LIN {X 0,Y 573.33,Z 232.072,A -85,B 0,C 180,E1 -2340.702,E2 -2340.702} C_VEL
LIN {X 0,Y 573.232,Z 232.084,A -85,B 0,C 180,E1 -2343.514,E2 -2343.514} C_VEL
LIN {X 0,Y 573.285,Z 232.078,A -85,B 0,C 180,E1 -2345.627,E2 -2345.627} C_VEL
LIN {X 0,Y 573.302,Z 232.075,A -85,B 0,C 180,E1 -2348.458,E2 -2348.458} C_VEL
LIN {X 0,Y 573.232,Z 232.085,A -85,B 0,C 180,E1 -2350.596,E2 -2350.596} C_VEL
LIN {X 0,Y 573.186,Z 234.19,A -85,B 0,C 180,E1 -2352.03,E2 -2352.03} C_VEL
LIN {X 0,Y 573.193,Z 239.014,A -85,B 0,C 180,E1 -2354.92,E2 -2354.92} C_VEL
LIN {X 0,Y 573.132,Z 244.034,A -85,B 0,C 180,E1 -2357.851,E2 -2357.851} C_VEL
LIN {X 0,Y 573.107,Z 249.239,A -85,B 0,C 180,E1 -2360.831,E2 -2360.831} C_VEL
LIN {X 0,Y 573.09,Z 253.122,A -85,B 0,C 180,E1 -2363.113,E2 -2363.113} C_VEL
LIN {X 0,Y 573.02,Z 254.947,A -85,B 0,C 180,E1 -2364.165,E2 -2364.165} C_VEL
LIN {X 0,Y 572.332,Z 256.016,A -85,B 0,C 180,E1 -2364.741,E2 -2364.741} C_VEL
LIN {X 0,Y 569.439,Z 257.913,A -85,B 0,C 180,E1 -2365.674,E2 -2365.674} C_VEL
LIN {X 0,Y 567.014,Z 259.45,A -85,B 0,C 180,E1 -2366.423,E2 -2366.423} C_VEL
LIN {X 0,Y 565.992,Z 260.576,A -85,B 0,C 180,E1 -2367.003,E2 -2367.003} C_VEL
LIN {X 0,Y 565.919,Z 260.939,A -85,B 0,C 180,E1 -2367.2,E2 -2367.2} C_VEL
LIN {X 0,Y 565.873,Z 265.731,A -85,B 0,C 180,E1 -2369.787,E2 -2369.787} C_VEL
LIN {X 0,Y 565.858,Z 270.593,A -85,B 0,C 180,E1 -2372.377,E2 -2372.377} C_VEL
LIN {X 0,Y 565.894,Z 272.598,A -85,B 0,C 180,E1 -2373.417,E2 -2373.417} C_VEL
LIN {X 0,Y 566.93,Z 280.016,A -85,B 0,C 180,E1 -2373.598,E2 -2373.598} C_VEL
LIN {X 0,Y 566.775,Z 292.555,A -85,B 0,C 180,E1 -2373.97,E2 -2373.97} C_VEL
LIN {X 0,Y 566.643,Z 304.455,A -85,B 0,C 180,E1 -2374.462,E2 -2374.462} C_VEL
LIN {X 0,Y 566.533,Z 315.205,A -85,B 0,C 180,E1 -2375.042,E2 -2375.042} C_VEL
LIN {X 0,Y 566.409,Z 325.926,A -85,B 0,C 180,E1 -2375.771,E2 -2375.771} C_VEL
LIN {X 0,Y 566.276,Z 336.609,A -85,B 0,C 180,E1 -2376.674,E2 -2376.674} C_VEL
LIN {X 0,Y 566.178,Z 344.253,A -85,B 0,C 180,E1 -2377.461,E2 -2377.461} C_VEL
LIN {X 0,Y 566.028,Z 352.881,A -85,B 0,C 180,E1 -2378.536,E2 -2378.536} C_VEL
LIN {X 0,Y 565.982,Z 360.04,A -85,B 0,C 180,E1 -2379.659,E2 -2379.659} C_VEL
LIN {X 0,Y 565.939,Z 365.613,A -85,B 0,C 180,E1 -2380.756,E2 -2380.756} C_VEL
LIN {X 0,Y 565.92,Z 369.886,A -85,B 0,C 180,E1 -2381.832,E2 -2381.832} C_VEL
LIN {X 0,Y 565.849,Z 373.537,A -85,B 0,C 180,E1 -2383.086,E2 -2383.086} C_VEL
LIN {X 0,Y 565.854,Z 375.448,A -85,B 0,C 180,E1 -2384.068,E2 -2384.068} C_VEL
LIN {X 0,Y 565.874,Z 376.606,A -85,B 0,C 180,E1 -2385.065,E2 -2385.065} C_VEL
LIN {X 0,Y 565.845,Z 376.997,A -85,B 0,C 180,E1 -2386.084,E2 -2386.084} C_VEL
LIN {X 0,Y 565.846,Z 376.542,A -85,B 0,C 180,E1 -2387.12,E2 -2387.12} C_VEL
LIN {X 0,Y 565.851,Z 375.204,A -85,B 0,C 180,E1 -2388.176,E2 -2388.176} C_VEL
LIN {X 0,Y 565.869,Z 372.917,A -85,B 0,C 180,E1 -2389.252,E2 -2389.252} C_VEL
LIN {X 0,Y 565.945,Z 369.582,A -85,B 0,C 180,E1 -2390.345,E2 -2390.345} C_VEL
LIN {X 0,Y 565.942,Z 364.323,A -85,B 0,C 180,E1 -2391.618,E2 -2391.618} C_VEL
LIN {X 0,Y 566.024,Z 357.686,A -85,B 0,C 180,E1 -2392.828,E2 -2392.828} C_VEL
LIN {X 0,Y 566.066,Z 351.029,A -85,B 0,C 180,E1 -2393.802,E2 -2393.802} C_VEL
LIN {X 0,Y 566.178,Z 342.022,A -85,B 0,C 180,E1 -2394.876,E2 -2394.876} C_VEL
LIN {X 0,Y 566.32,Z 331.919,A -85,B 0,C 180,E1 -2395.838,E2 -2395.838} C_VEL
LIN {X 0,Y 566.432,Z 320.626,A -85,B 0,C 180,E1 -2396.7,E2 -2396.7} C_VEL
LIN {X 0,Y 566.531,Z 308.684,A -85,B 0,C 180,E1 -2397.416,E2 -2397.416} C_VEL
LIN {X 0,Y 566.702,Z 296.228,A -85,B 0,C 180,E1 -2397.984,E2 -2397.984} C_VEL
LIN {X 0,Y 566.865,Z 283.269,A -85,B 0,C 180,E1 -2398.412,E2 -2398.412} C_VEL
LIN {X 0,Y 566.692,Z 277.469,A -85,B 0,C 180,E1 -2398.558,E2 -2398.558} C_VEL
LIN {X 0,Y 565.854,Z 272.554,A -85,B 0,C 180,E1 -2398.677,E2 -2398.677} C_VEL
LIN {X 0,Y 565.849,Z 268.118,A -85,B 0,C 180,E1 -2401.028,E2 -2401.028} C_VEL
LIN {X 0,Y 565.887,Z 263.61,A -85,B 0,C 180,E1 -2403.443,E2 -2403.443} C_VEL
LIN {X 0,Y 565.906,Z 259.28,A -85,B 0,C 180,E1 -2405.807,E2 -2405.807} C_VEL
LIN {X 0,Y 565.967,Z 254.293,A -85,B 0,C 180,E1 -2408.639,E2 -2408.639} C_VEL
LIN {X 0,Y 566.028,Z 249.915,A -85,B 0,C 180,E1 -2411.167,E2 -2411.167} C_VEL
LIN {X 0,Y 566.041,Z 244.734,A -85,B 0,C 180,E1 -2414.148,E2 -2414.148} C_VEL
LIN {X 0,Y 566.11,Z 239.77,A -85,B 0,C 180,E1 -2417.088,E2 -2417.088} C_VEL
LIN {X 0,Y 566.19,Z 236.152,A -85,B 0,C 180,E1 -2419.27,E2 -2419.27} C_VEL
LIN {X 0,Y 566.131,Z 233.791,A -85,B 0,C 180,E1 -2420.713,E2 -2420.713} C_VEL
LIN {X 0,Y 566.158,Z 232.962,A -85,B 0,C 180,E1 -2421.434,E2 -2421.434} C_VEL
LIN {X 0,Y 566.197,Z 232.961,A -85,B 0,C 180,E1 -2423.586,E2 -2423.586} C_VEL
LIN {X 0,Y 566.184,Z 232.96,A -85,B 0,C 180,E1 -2425.729,E2 -2425.729} C_VEL
LIN {X 0,Y 566.267,Z 232.949,A -85,B 0,C 180,E1 -2427.866,E2 -2427.866} C_VEL
LIN {X 0,Y 566.297,Z 232.948,A -85,B 0,C 180,E1 -2430.711,E2 -2430.711} C_VEL
LIN {X 0,Y 566.267,Z 232.95,A -85,B 0,C 180,E1 -2432.846,E2 -2432.846} C_VEL
LIN {X 0,Y 566.251,Z 232.954,A -85,B 0,C 180,E1 -2435.698,E2 -2435.698} C_VEL
LIN {X 0,Y 566.241,Z 232.953,A -85,B 0,C 180,E1 -2438.565,E2 -2438.565} C_VEL
LIN {X 0,Y 566.24,Z 232.954,A -85,B 0,C 180,E1 -2441.454,E2 -2441.454} C_VEL
LIN {X 0,Y 566.223,Z 232.955,A -85,B 0,C 180,E1 -2444.507,E2 -2444.507} C_VEL
LIN {X 0,Y 566.195,Z 232.959,A -85,B 0,C 180,E1 -2447.332,E2 -2447.332} C_VEL
LIN {X 0,Y 566.21,Z 232.957,A -85,B 0,C 180,E1 -2450.337,E2 -2450.337} C_VEL
LIN {X 0,Y 566.22,Z 232.956,A -85,B 0,C 180,E1 -2453.402,E2 -2453.402} C_VEL
LIN {X 0,Y 566.213,Z 232.957,A -85,B 0,C 180,E1 -2455.749,E2 -2455.749} C_VEL
LIN {X 0,Y 566.198,Z 232.96,A -85,B 0,C 180,E1 -2458.204,E2 -2458.204} C_VEL
LIN {X 0,Y 566.184,Z 232.961,A -85,B 0,C 180,E1 -2460.592,E2 -2460.592} C_VEL
LIN {X 0,Y 566.218,Z 232.957,A -85,B 0,C 180,E1 -2463.102,E2 -2463.102} C_VEL
LIN {X 0,Y 566.201,Z 232.96,A -85,B 0,C 180,E1 -2465.689,E2 -2465.689} C_VEL
LIN {X 0,Y 566.207,Z 232.956,A -85,B 0,C 180,E1 -2468.56,E2 -2468.56} C_VEL
LIN {X 0,Y 566.201,Z 232.958,A -85,B 0,C 180,E1 -2471.136,E2 -2471.136} C_VEL
LIN {X 0,Y 566.189,Z 232.962,A -85,B 0,C 180,E1 -2474.036,E2 -2474.036} C_VEL
LIN {X 0,Y 566.202,Z 232.957,A -85,B 0,C 180,E1 -2477.082,E2 -2477.082} C_VEL
LIN {X 0,Y 566.216,Z 232.957,A -85,B 0,C 180,E1 -2479.803,E2 -2479.803} C_VEL
LIN {X 0,Y 566.188,Z 232.961,A -85,B 0,C 180,E1 -2482.599,E2 -2482.599} C_VEL
LIN {X 0,Y 566.209,Z 232.957,A -85,B 0,C 180,E1 -2485.184,E2 -2485.184} C_VEL
LIN {X 0,Y 566.225,Z 232.954,A -85,B 0,C 180,E1 -2487.744,E2 -2487.744} C_VEL
LIN {X 0,Y 566.217,Z 232.955,A -85,B 0,C 180,E1 -2490.324,E2 -2490.324} C_VEL
LIN {X 0,Y 566.225,Z 232.956,A -85,B 0,C 180,E1 -2493.336,E2 -2493.336} C_VEL
LIN {X 0,Y 566.19,Z 232.96,A -85,B 0,C 180,E1 -2495.82,E2 -2495.82} C_VEL
LIN {X 0,Y 566.208,Z 232.958,A -85,B 0,C 180,E1 -2498.903,E2 -2498.903} C_VEL
LIN {X 0,Y 566.204,Z 232.957,A -85,B 0,C 180,E1 -2501.173,E2 -2501.173} C_VEL
LIN {X 0,Y 566.213,Z 232.956,A -85,B 0,C 180,E1 -2503.413,E2 -2503.413} C_VEL
LIN {X 0,Y 566.189,Z 232.962,A -85,B 0,C 180,E1 -2506.36,E2 -2506.36} C_VEL
LIN {X 0,Y 566.267,Z 232.951,A -85,B 0,C 180,E1 -2508.655,E2 -2508.655} C_VEL
LIN {X 0,Y 566.242,Z 232.954,A -85,B 0,C 180,E1 -2511.435,E2 -2511.435} C_VEL
LIN {X 0,Y 566.252,Z 232.951,A -85,B 0,C 180,E1 -2514.303,E2 -2514.303} C_VEL
LIN {X 0,Y 566.275,Z 232.948,A -85,B 0,C 180,E1 -2517.867,E2 -2517.867} C_VEL
LIN {X 0,Y 566.3,Z 232.948,A -85,B 0,C 180,E1 -2520.712,E2 -2520.712} C_VEL
LIN {X 0,Y 566.264,Z 232.95,A -85,B 0,C 180,E1 -2522.846,E2 -2522.846} C_VEL
LIN {X 0,Y 566.253,Z 232.954,A -85,B 0,C 180,E1 -2525.699,E2 -2525.699} C_VEL
LIN {X 0,Y 566.223,Z 232.955,A -85,B 0,C 180,E1 -2528.567,E2 -2528.567} C_VEL
LIN {X 0,Y 566.236,Z 232.954,A -85,B 0,C 180,E1 -2531.455,E2 -2531.455} C_VEL
LIN {X 0,Y 566.229,Z 232.954,A -85,B 0,C 180,E1 -2534.508,E2 -2534.508} C_VEL
LIN {X 0,Y 566.195,Z 232.959,A -85,B 0,C 180,E1 -2537.332,E2 -2537.332} C_VEL
LIN {X 0,Y 566.209,Z 232.957,A -85,B 0,C 180,E1 -2540.338,E2 -2540.338} C_VEL
LIN {X 0,Y 566.185,Z 232.961,A -85,B 0,C 180,E1 -2543.405,E2 -2543.405} C_VEL
LIN {X 0,Y 566.21,Z 232.958,A -85,B 0,C 180,E1 -2545.75,E2 -2545.75} C_VEL
LIN {X 0,Y 566.205,Z 232.959,A -85,B 0,C 180,E1 -2548.204,E2 -2548.204} C_VEL
LIN {X 0,Y 566.192,Z 232.96,A -85,B 0,C 180,E1 -2551.078,E2 -2551.078} C_VEL
LIN {X 0,Y 566.195,Z 232.958,A -85,B 0,C 180,E1 -2553.733,E2 -2553.733} C_VEL
LIN {X 0,Y 566.206,Z 232.958,A -85,B 0,C 180,E1 -2556.57,E2 -2556.57} C_VEL
LIN {X 0,Y 566.21,Z 232.956,A -85,B 0,C 180,E1 -2559.686,E2 -2559.686} C_VEL
LIN {X 0,Y 566.187,Z 232.959,A -85,B 0,C 180,E1 -2562.09,E2 -2562.09} C_VEL
LIN {X 0,Y 566.167,Z 232.963,A -85,B 0,C 180,E1 -2565.037,E2 -2565.037} C_VEL
LIN {X 0,Y 566.211,Z 232.957,A -85,B 0,C 180,E1 -2567.913,E2 -2567.913} C_VEL
LIN {X 0,Y 566.22,Z 232.955,A -85,B 0,C 180,E1 -2570.728,E2 -2570.728} C_VEL
LIN {X 0,Y 566.237,Z 233.104,A -85,B 0,C 180,E1 -2573.535,E2 -2573.535} C_VEL
LIN {X 0,Y 566.579,Z 236.582,A -85,B 0,C 180,E1 -2574.954,E2 -2574.954} C_VEL
LIN {X 0,Y 566.458,Z 243.827,A -85,B 0,C 180,E1 -2577.759,E2 -2577.759} C_VEL
LIN {X 0,Y 566.355,Z 250.603,A -85,B 0,C 180,E1 -2580.302,E2 -2580.302} C_VEL
LIN {X 0,Y 566.227,Z 257.034,A -85,B 0,C 180,E1 -2582.662,E2 -2582.662} C_VEL
LIN {X 0,Y 566.18,Z 264.979,A -85,B 0,C 180,E1 -2585.428,E2 -2585.428} C_VEL
LIN {X 0,Y 566.172,Z 272.923,A -85,B 0,C 180,E1 -2588.137,E2 -2588.137} C_VEL
LIN {X 0,Y 566.119,Z 280.374,A -85,B 0,C 180,E1 -2590.647,E2 -2590.647} C_VEL
LIN {X 0,Y 566.058,Z 289.71,A -85,B 0,C 180,E1 -2593.779,E2 -2593.779} C_VEL
LIN {X 0,Y 565.998,Z 298.614,A -85,B 0,C 180,E1 -2596.72,E2 -2596.72} C_VEL
LIN {X 0,Y 565.983,Z 300.492,A -85,B 0,C 180,E1 -2597.336,E2 -2597.336} C_VEL
LIN {X 0,Y 566.955,Z 307.515,A -85,B 0,C 180,E1 -2597.494,E2 -2597.494} C_VEL
LIN {X 0,Y 566.829,Z 319.879,A -85,B 0,C 180,E1 -2597.832,E2 -2597.832} C_VEL
LIN {X 0,Y 566.67,Z 331.612,A -85,B 0,C 180,E1 -2598.287,E2 -2598.287} C_VEL
LIN {X 0,Y 566.551,Z 342.937,A -85,B 0,C 180,E1 -2598.866,E2 -2598.866} C_VEL
LIN {X 0,Y 566.431,Z 353.485,A -85,B 0,C 180,E1 -2599.545,E2 -2599.545} C_VEL
LIN {X 0,Y 566.301,Z 363.648,A -85,B 0,C 180,E1 -2600.355,E2 -2600.355} C_VEL
LIN {X 0,Y 566.166,Z 372.787,A -85,B 0,C 180,E1 -2601.254,E2 -2601.254} C_VEL
LIN {X 0,Y 566.081,Z 381.689,A -85,B 0,C 180,E1 -2602.33,E2 -2602.33} C_VEL
LIN {X 0,Y 565.968,Z 388.956,A -85,B 0,C 180,E1 -2603.422,E2 -2603.422} C_VEL
LIN {X 0,Y 566.004,Z 393.68,A -85,B 0,C 180,E1 -2604.299,E2 -2604.299} C_VEL
LIN {X 0,Y 565.933,Z 398.372,A -85,B 0,C 180,E1 -2605.37,E2 -2605.37} C_VEL
LIN {X 0,Y 565.927,Z 401.957,A -85,B 0,C 180,E1 -2606.44,E2 -2606.44} C_VEL
LIN {X 0,Y 565.878,Z 403.808,A -85,B 0,C 180,E1 -2607.152,E2 -2607.152} C_VEL
LIN {X 0,Y 565.846,Z 406.185,A -85,B 0,C 180,E1 -2608.577,E2 -2608.577} C_VEL
LIN {X 0,Y 565.839,Z 407,A -85,B 0,C 180,E1 -2610,E2 -2610} C_VEL
LIN {X 0,Y 565.846,Z 406.186,A -85,B 0,C 180,E1 -2611.423,E2 -2611.423} C_VEL
LIN {X 0,Y 565.878,Z 403.81,A -85,B 0,C 180,E1 -2612.847,E2 -2612.847} C_VEL
LIN {X 0,Y 565.926,Z 400.896,A -85,B 0,C 180,E1 -2613.916,E2 -2613.916} C_VEL
LIN {X 0,Y 565.878,Z 396.95,A -85,B 0,C 180,E1 -2614.987,E2 -2614.987} C_VEL
LIN {X 0,Y 566.002,Z 391.868,A -85,B 0,C 180,E1 -2616.058,E2 -2616.058} C_VEL
LIN {X 0,Y 566.04,Z 385.47,A -85,B 0,C 180,E1 -2617.132,E2 -2617.132} C_VEL
LIN {X 0,Y 566.134,Z 377.48,A -85,B 0,C 180,E1 -2618.207,E2 -2618.207} C_VEL
LIN {X 0,Y 566.229,Z 369.338,A -85,B 0,C 180,E1 -2619.105,E2 -2619.105} C_VEL
LIN {X 0,Y 566.349,Z 359.404,A -85,B 0,C 180,E1 -2620.004,E2 -2620.004} C_VEL
LIN {X 0,Y 566.502,Z 348.338,A -85,B 0,C 180,E1 -2620.805,E2 -2620.805} C_VEL
LIN {X 0,Y 566.609,Z 335.952,A -85,B 0,C 180,E1 -2621.51,E2 -2621.51} C_VEL
LIN {X 0,Y 566.777,Z 323.777,A -85,B 0,C 180,E1 -2622.032,E2 -2622.032} C_VEL
LIN {X 0,Y 566.916,Z 310.361,A -85,B 0,C 180,E1 -2622.438,E2 -2622.438} C_VEL
LIN {X 0,Y 566.646,Z 304.829,A -85,B 0,C 180,E1 -2622.566,E2 -2622.566} C_VEL
LIN {X 0,Y 565.983,Z 300.493,A -85,B 0,C 180,E1 -2622.664,E2 -2622.664} C_VEL
LIN {X 0,Y 566.029,Z 291.936,A -85,B 0,C 180,E1 -2625.482,E2 -2625.482} C_VEL
LIN {X 0,Y 566.089,Z 283.032,A -85,B 0,C 180,E1 -2628.456,E2 -2628.456} C_VEL
LIN {X 0,Y 566.161,Z 274.238,A -85,B 0,C 180,E1 -2631.407,E2 -2631.407} C_VEL
LIN {X 0,Y 566.199,Z 265.985,A -85,B 0,C 180,E1 -2634.18,E2 -2634.18} C_VEL
LIN {X 0,Y 566.194,Z 258.877,A -85,B 0,C 180,E1 -2636.655,E2 -2636.655} C_VEL
LIN {X 0,Y 566.315,Z 251.547,A -85,B 0,C 180,E1 -2639.32,E2 -2639.32} C_VEL
LIN {X 0,Y 566.404,Z 245.911,A -85,B 0,C 180,E1 -2641.408,E2 -2641.408} C_VEL
LIN {X 0,Y 566.493,Z 239.335,A -85,B 0,C 180,E1 -2643.936,E2 -2643.936} C_VEL
LIN {X 0,Y 566.548,Z 235.025,A -85,B 0,C 180,E1 -2645.663,E2 -2645.663} C_VEL
LIN {X 0,Y 566.249,Z 232.955,A -85,B 0,C 180,E1 -2646.565,E2 -2646.565} C_VEL
LIN {X 0,Y 566.214,Z 232.958,A -85,B 0,C 180,E1 -2649.685,E2 -2649.685} C_VEL
LIN {X 0,Y 566.213,Z 232.958,A -85,B 0,C 180,E1 -2652.086,E2 -2652.086} C_VEL
LIN {X 0,Y 566.171,Z 232.962,A -85,B 0,C 180,E1 -2655.035,E2 -2655.035} C_VEL
LIN {X 0,Y 566.216,Z 232.957,A -85,B 0,C 180,E1 -2658.135,E2 -2658.135} C_VEL
LIN {X 0,Y 566.219,Z 232.958,A -85,B 0,C 180,E1 -2660.726,E2 -2660.726} C_VEL
LIN {X 0,Y 566.215,Z 232.958,A -85,B 0,C 180,E1 -2663.782,E2 -2663.782} C_VEL
LIN {X 0,Y 566.208,Z 232.958,A -85,B 0,C 180,E1 -2666.265,E2 -2666.265} C_VEL
LIN {X 0,Y 566.2,Z 232.96,A -85,B 0,C 180,E1 -2668.92,E2 -2668.92} C_VEL
LIN {X 0,Y 566.19,Z 232.961,A -85,B 0,C 180,E1 -2671.046,E2 -2671.046} C_VEL
LIN {X 0,Y 566.213,Z 232.957,A -85,B 0,C 180,E1 -2673.458,E2 -2673.458} C_VEL
LIN {X 0,Y 566.194,Z 232.961,A -85,B 0,C 180,E1 -2675.818,E2 -2675.818} C_VEL
LIN {X 0,Y 566.202,Z 232.96,A -85,B 0,C 180,E1 -2678.901,E2 -2678.901} C_VEL
LIN {X 0,Y 566.207,Z 232.96,A -85,B 0,C 180,E1 -2681.172,E2 -2681.172} C_VEL
LIN {X 0,Y 566.214,Z 232.957,A -85,B 0,C 180,E1 -2683.412,E2 -2683.412} C_VEL
LIN {X 0,Y 566.196,Z 232.961,A -85,B 0,C 180,E1 -2686.358,E2 -2686.358} C_VEL
LIN {X 0,Y 566.268,Z 232.95,A -85,B 0,C 180,E1 -2688.653,E2 -2688.653} C_VEL
LIN {X 0,Y 566.244,Z 232.955,A -85,B 0,C 180,E1 -2691.434,E2 -2691.434} C_VEL
LIN {X 0,Y 566.255,Z 232.953,A -85,B 0,C 180,E1 -2694.301,E2 -2694.301} C_VEL
LIN {X 0,Y 566.272,Z 232.95,A -85,B 0,C 180,E1 -2697.865,E2 -2697.865} C_VEL
LIN {X 0,Y 566.299,Z 232.948,A -85,B 0,C 180,E1 -2700.71,E2 -2700.71} C_VEL
LIN {X 0,Y 566.271,Z 232.951,A -85,B 0,C 180,E1 -2702.845,E2 -2702.845} C_VEL
LIN {X 0,Y 566.254,Z 232.954,A -85,B 0,C 180,E1 -2705.697,E2 -2705.697} C_VEL
LIN {X 0,Y 566.242,Z 232.954,A -85,B 0,C 180,E1 -2708.565,E2 -2708.565} C_VEL
LIN {X 0,Y 566.166,Z 232.966,A -85,B 0,C 180,E1 -2710.73,E2 -2710.73} C_VEL
LIN {X 0,Y 566.133,Z 237.694,A -85,B 0,C 180,E1 -2713.642,E2 -2713.642} C_VEL
LIN {X 0,Y 566.097,Z 241.361,A -85,B 0,C 180,E1 -2715.849,E2 -2715.849} C_VEL
LIN {X 0,Y 566.06,Z 245.161,A -85,B 0,C 180,E1 -2718.082,E2 -2718.082} C_VEL
LIN {X 0,Y 566.058,Z 250.432,A -85,B 0,C 180,E1 -2721.102,E2 -2721.102} C_VEL
LIN {X 0,Y 565.998,Z 254.327,A -85,B 0,C 180,E1 -2723.411,E2 -2723.411} C_VEL
LIN {X 0,Y 565.943,Z 258.382,A -85,B 0,C 180,E1 -2725.761,E2 -2725.761} C_VEL
LIN {X 0,Y 565.919,Z 260.939,A -85,B 0,C 180,E1 -2727.2,E2 -2727.2} C_VEL
LIN {X 0,Y 565.273,Z 262.049,A -85,B 0,C 180,E1 -2727.783,E2 -2727.783} C_VEL
LIN {X 0,Y 562.401,Z 263.962,A -85,B 0,C 180,E1 -2728.726,E2 -2728.726} C_VEL
LIN {X 0,Y 559.946,Z 265.502,A -85,B 0,C 180,E1 -2729.485,E2 -2729.485} C_VEL
LIN {X 0,Y 558.875,Z 266.643,A -85,B 0,C 180,E1 -2730.072,E2 -2730.072} C_VEL
LIN {X 0,Y 558.78,Z 267.016,A -85,B 0,C 180,E1 -2730.272,E2 -2730.272} C_VEL
LIN {X 0,Y 558.806,Z 272.547,A -85,B 0,C 180,E1 -2733.247,E2 -2733.247} C_VEL
LIN {X 0,Y 560.006,Z 280.292,A -85,B 0,C 180,E1 -2733.449,E2 -2733.449} C_VEL
LIN {X 0,Y 559.841,Z 291.874,A -85,B 0,C 180,E1 -2733.794,E2 -2733.794} C_VEL
LIN {X 0,Y 559.686,Z 304.064,A -85,B 0,C 180,E1 -2734.298,E2 -2734.298} C_VEL
LIN {X 0,Y 559.529,Z 316.156,A -85,B 0,C 180,E1 -2734.964,E2 -2734.964} C_VEL
LIN {X 0,Y 559.367,Z 327.305,A -85,B 0,C 180,E1 -2735.748,E2 -2735.748} C_VEL
LIN {X 0,Y 559.229,Z 336.837,A -85,B 0,C 180,E1 -2736.576,E2 -2736.576} C_VEL
LIN {X 0,Y 559.128,Z 345.561,A -85,B 0,C 180,E1 -2737.5,E2 -2737.5} C_VEL
LIN {X 0,Y 558.974,Z 353.928,A -85,B 0,C 180,E1 -2738.595,E2 -2738.595} C_VEL
LIN {X 0,Y 558.898,Z 360.464,A -85,B 0,C 180,E1 -2739.654,E2 -2739.654} C_VEL
LIN {X 0,Y 558.842,Z 366.282,A -85,B 0,C 180,E1 -2740.839,E2 -2740.839} C_VEL
LIN {X 0,Y 558.817,Z 370.953,A -85,B 0,C 180,E1 -2742.098,E2 -2742.098} C_VEL
LIN {X 0,Y 558.761,Z 373.797,A -85,B 0,C 180,E1 -2743.156,E2 -2743.156} C_VEL
LIN {X 0,Y 558.771,Z 375.69,A -85,B 0,C 180,E1 -2744.2,E2 -2744.2} C_VEL
LIN {X 0,Y 558.782,Z 376.721,A -85,B 0,C 180,E1 -2745.226,E2 -2745.226} C_VEL
LIN {X 0,Y 558.753,Z 376.966,A -85,B 0,C 180,E1 -2746.229,E2 -2746.229} C_VEL
LIN {X 0,Y 558.743,Z 376.475,A -85,B 0,C 180,E1 -2747.218,E2 -2747.218} C_VEL
LIN {X 0,Y 558.755,Z 375.218,A -85,B 0,C 180,E1 -2748.193,E2 -2748.193} C_VEL
LIN {X 0,Y 558.781,Z 373.256,A -85,B 0,C 180,E1 -2749.155,E2 -2749.155} C_VEL
LIN {X 0,Y 558.862,Z 368.976,A -85,B 0,C 180,E1 -2750.576,E2 -2750.576} C_VEL
LIN {X 0,Y 558.864,Z 364.744,A -85,B 0,C 180,E1 -2751.596,E2 -2751.596} C_VEL
LIN {X 0,Y 558.907,Z 359.361,A -85,B 0,C 180,E1 -2752.634,E2 -2752.634} C_VEL
LIN {X 0,Y 559.001,Z 351.932,A -85,B 0,C 180,E1 -2753.78,E2 -2753.78} C_VEL
LIN {X 0,Y 559.129,Z 343.832,A -85,B 0,C 180,E1 -2754.785,E2 -2754.785} C_VEL
LIN {X 0,Y 559.247,Z 334.904,A -85,B 0,C 180,E1 -2755.695,E2 -2755.695} C_VEL
LIN {X 0,Y 559.393,Z 324.634,A -85,B 0,C 180,E1 -2756.55,E2 -2756.55} C_VEL
LIN {X 0,Y 559.529,Z 313.122,A -85,B 0,C 180,E1 -2757.31,E2 -2757.31} C_VEL
LIN {X 0,Y 559.662,Z 301.651,A -85,B 0,C 180,E1 -2757.905,E2 -2757.905} C_VEL
LIN {X 0,Y 559.874,Z 289.908,A -85,B 0,C 180,E1 -2758.365,E2 -2758.365} C_VEL
LIN {X 0,Y 559.844,Z 278.851,A -85,B 0,C 180,E1 -2758.681,E2 -2758.681} C_VEL
LIN {X 0,Y 558.784,Z 272.55,A -85,B 0,C 180,E1 -2758.842,E2 -2758.842} C_VEL
LIN {X 0,Y 558.769,Z 267.25,A -85,B 0,C 180,E1 -2761.692,E2 -2761.692} C_VEL
LIN {X 0,Y 558.786,Z 263.256,A -85,B 0,C 180,E1 -2763.884,E2 -2763.884} C_VEL
LIN {X 0,Y 558.857,Z 258.396,A -85,B 0,C 180,E1 -2766.635,E2 -2766.635} C_VEL
LIN {X 0,Y 558.918,Z 253.644,A -85,B 0,C 180,E1 -2769.386,E2 -2769.386} C_VEL
LIN {X 0,Y 558.942,Z 249.668,A -85,B 0,C 180,E1 -2771.679,E2 -2771.679} C_VEL
LIN {X 0,Y 558.972,Z 245.784,A -85,B 0,C 180,E1 -2773.943,E2 -2773.943} C_VEL
LIN {X 0,Y 559.054,Z 240.803,A -85,B 0,C 180,E1 -2776.922,E2 -2776.922} C_VEL
LIN {X 0,Y 559.13,Z 237.184,A -85,B 0,C 180,E1 -2779.133,E2 -2779.133} C_VEL
LIN {X 0,Y 559.088,Z 233.843,A -85,B 0,C 180,E1 -2781.324,E2 -2781.324} C_VEL
LIN {X 0,Y 559.16,Z 233.837,A -85,B 0,C 180,E1 -2783.505,E2 -2783.505} C_VEL
LIN {X 0,Y 559.143,Z 233.837,A -85,B 0,C 180,E1 -2785.675,E2 -2785.675} C_VEL
LIN {X 0,Y 559.239,Z 233.824,A -85,B 0,C 180,E1 -2787.84,E2 -2787.84} C_VEL
LIN {X 0,Y 559.267,Z 233.824,A -85,B 0,C 180,E1 -2790.72,E2 -2790.72} C_VEL
LIN {X 0,Y 559.234,Z 233.826,A -85,B 0,C 180,E1 -2792.881,E2 -2792.881} C_VEL
LIN {X 0,Y 559.22,Z 233.829,A -85,B 0,C 180,E1 -2795.77,E2 -2795.77} C_VEL
LIN {X 0,Y 559.195,Z 233.83,A -85,B 0,C 180,E1 -2798.674,E2 -2798.674} C_VEL
LIN {X 0,Y 559.199,Z 233.832,A -85,B 0,C 180,E1 -2801.6,E2 -2801.6} C_VEL
LIN {X 0,Y 559.188,Z 233.831,A -85,B 0,C 180,E1 -2804.596,E2 -2804.596} C_VEL
LIN {X 0,Y 559.154,Z 233.838,A -85,B 0,C 180,E1 -2807.557,E2 -2807.557} C_VEL
LIN {X 0,Y 559.165,Z 233.836,A -85,B 0,C 180,E1 -2809.837,E2 -2809.837} C_VEL
LIN {X 0,Y 559.145,Z 233.838,A -85,B 0,C 180,E1 -2812.152,E2 -2812.152} C_VEL
LIN {X 0,Y 559.15,Z 233.837,A -85,B 0,C 180,E1 -2814.505,E2 -2814.505} C_VEL
LIN {X 0,Y 559.17,Z 233.834,A -85,B 0,C 180,E1 -2816.902,E2 -2816.902} C_VEL
LIN {X 0,Y 559.179,Z 233.834,A -85,B 0,C 180,E1 -2819.865,E2 -2819.865} C_VEL
LIN {X 0,Y 559.165,Z 233.833,A -85,B 0,C 180,E1 -2822.714,E2 -2822.714} C_VEL
LIN {X 0,Y 559.146,Z 233.837,A -85,B 0,C 180,E1 -2825.322,E2 -2825.322} C_VEL
LIN {X 0,Y 559.125,Z 233.842,A -85,B 0,C 180,E1 -2828.017,E2 -2828.017} C_VEL
LIN {X 0,Y 559.165,Z 233.834,A -85,B 0,C 180,E1 -2830.811,E2 -2830.811} C_VEL
LIN {X 0,Y 559.153,Z 233.837,A -85,B 0,C 180,E1 -2833.732,E2 -2833.732} C_VEL
LIN {X 0,Y 559.161,Z 233.835,A -85,B 0,C 180,E1 -2836.801,E2 -2836.801} C_VEL
LIN {X 0,Y 559.165,Z 233.835,A -85,B 0,C 180,E1 -2839.19,E2 -2839.19} C_VEL
LIN {X 0,Y 559.125,Z 233.839,A -85,B 0,C 180,E1 -2841.983,E2 -2841.983} C_VEL
LIN {X 0,Y 559.147,Z 233.838,A -85,B 0,C 180,E1 -2844.679,E2 -2844.679} C_VEL
LIN {X 0,Y 559.164,Z 233.836,A -85,B 0,C 180,E1 -2847.362,E2 -2847.362} C_VEL
LIN {X 0,Y 559.178,Z 233.832,A -85,B 0,C 180,E1 -2850.136,E2 -2850.136} C_VEL
LIN {X 0,Y 559.172,Z 233.836,A -85,B 0,C 180,E1 -2853.17,E2 -2853.17} C_VEL
LIN {X 0,Y 559.148,Z 233.839,A -85,B 0,C 180,E1 -2855.496,E2 -2855.496} C_VEL
LIN {X 0,Y 559.167,Z 233.834,A -85,B 0,C 180,E1 -2858.625,E2 -2858.625} C_VEL
LIN {X 0,Y 559.162,Z 233.834,A -85,B 0,C 180,E1 -2860.927,E2 -2860.927} C_VEL
LIN {X 0,Y 559.162,Z 233.836,A -85,B 0,C 180,E1 -2863.949,E2 -2863.949} C_VEL
LIN {X 0,Y 559.163,Z 233.835,A -85,B 0,C 180,E1 -2866.185,E2 -2866.185} C_VEL
LIN {X 0,Y 559.204,Z 233.829,A -85,B 0,C 180,E1 -2869.135,E2 -2869.135} C_VEL
LIN {X 0,Y 559.202,Z 233.83,A -85,B 0,C 180,E1 -2872.055,E2 -2872.055} C_VEL
LIN {X 0,Y 559.25,Z 233.825,A -85,B 0,C 180,E1 -2874.954,E2 -2874.954} C_VEL
LIN {X 0,Y 559.246,Z 233.824,A -85,B 0,C 180,E1 -2877.84,E2 -2877.84} C_VEL
LIN {X 0,Y 559.27,Z 233.824,A -85,B 0,C 180,E1 -2880.721,E2 -2880.721} C_VEL
LIN {X 0,Y 559.232,Z 233.826,A -85,B 0,C 180,E1 -2882.882,E2 -2882.882} C_VEL
LIN {X 0,Y 559.222,Z 233.829,A -85,B 0,C 180,E1 -2885.771,E2 -2885.771} C_VEL
LIN {X 0,Y 559.182,Z 233.832,A -85,B 0,C 180,E1 -2888.675,E2 -2888.675} C_VEL
LIN {X 0,Y 559.2,Z 233.832,A -85,B 0,C 180,E1 -2891.601,E2 -2891.601} C_VEL
LIN {X 0,Y 559.194,Z 233.83,A -85,B 0,C 180,E1 -2894.596,E2 -2894.596} C_VEL
LIN {X 0,Y 559.155,Z 233.838,A -85,B 0,C 180,E1 -2897.558,E2 -2897.558} C_VEL
LIN {X 0,Y 559.167,Z 233.835,A -85,B 0,C 180,E1 -2899.838,E2 -2899.838} C_VEL
LIN {X 0,Y 559.137,Z 233.839,A -85,B 0,C 180,E1 -2902.154,E2 -2902.154} C_VEL
LIN {X 0,Y 559.175,Z 233.833,A -85,B 0,C 180,E1 -2905.188,E2 -2905.188} C_VEL
LIN {X 0,Y 559.189,Z 233.831,A -85,B 0,C 180,E1 -2907.712,E2 -2907.712} C_VEL
LIN {X 0,Y 559.156,Z 233.837,A -85,B 0,C 180,E1 -2911.02,E2 -2911.02} C_VEL
LIN {X 0,Y 559.155,Z 233.835,A -85,B 0,C 180,E1 -2913.949,E2 -2913.949} C_VEL
LIN {X 0,Y 559.157,Z 233.835,A -85,B 0,C 180,E1 -2916.448,E2 -2916.448} C_VEL
LIN {X 0,Y 559.177,Z 233.833,A -85,B 0,C 180,E1 -2918.935,E2 -2918.935} C_VEL
LIN {X 0,Y 559.164,Z 233.836,A -85,B 0,C 180,E1 -2921.771,E2 -2921.771} C_VEL
LIN {X 0,Y 559.135,Z 233.838,A -85,B 0,C 180,E1 -2924.74,E2 -2924.74} C_VEL
LIN {X 0,Y 559.174,Z 233.834,A -85,B 0,C 180,E1 -2927.864,E2 -2927.864} C_VEL
LIN {X 0,Y 559.181,Z 233.834,A -85,B 0,C 180,E1 -2930.135,E2 -2930.135} C_VEL
LIN {X 0,Y 559.201,Z 233.913,A -85,B 0,C 180,E1 -2933.342,E2 -2933.342} C_VEL
LIN {X 0,Y 559.563,Z 237.247,A -85,B 0,C 180,E1 -2934.725,E2 -2934.725} C_VEL
LIN {X 0,Y 559.491,Z 243.813,A -85,B 0,C 180,E1 -2937.312,E2 -2937.312} C_VEL
LIN {X 0,Y 559.358,Z 251.136,A -85,B 0,C 180,E1 -2940.106,E2 -2940.106} C_VEL
LIN {X 0,Y 559.173,Z 259.2,A -85,B 0,C 180,E1 -2943.098,E2 -2943.098} C_VEL
LIN {X 0,Y 559.154,Z 267.139,A -85,B 0,C 180,E1 -2945.89,E2 -2945.89} C_VEL
LIN {X 0,Y 559.088,Z 276.212,A -85,B 0,C 180,E1 -2949.007,E2 -2949.007} C_VEL
LIN {X 0,Y 559.021,Z 284.13,A -85,B 0,C 180,E1 -2951.682,E2 -2951.682} C_VEL
LIN {X 0,Y 558.968,Z 291.936,A -85,B 0,C 180,E1 -2954.317,E2 -2954.317} C_VEL
LIN {X 0,Y 558.925,Z 300.492,A -85,B 0,C 180,E1 -2957.173,E2 -2957.173} C_VEL
LIN {X 0,Y 560.015,Z 308.526,A -85,B 0,C 180,E1 -2957.36,E2 -2957.36} C_VEL
LIN {X 0,Y 559.878,Z 321.309,A -85,B 0,C 180,E1 -2957.729,E2 -2957.729} C_VEL
LIN {X 0,Y 559.723,Z 332.283,A -85,B 0,C 180,E1 -2958.171,E2 -2958.171} C_VEL
LIN {X 0,Y 559.57,Z 343.696,A -85,B 0,C 180,E1 -2958.769,E2 -2958.769} C_VEL
LIN {X 0,Y 559.428,Z 354.746,A -85,B 0,C 180,E1 -2959.504,E2 -2959.504} C_VEL
LIN {X 0,Y 559.244,Z 365.6,A -85,B 0,C 180,E1 -2960.415,E2 -2960.415} C_VEL
LIN {X 0,Y 559.127,Z 374.413,A -85,B 0,C 180,E1 -2961.325,E2 -2961.325} C_VEL
LIN {X 0,Y 558.997,Z 383.003,A -85,B 0,C 180,E1 -2962.414,E2 -2962.414} C_VEL
LIN {X 0,Y 558.885,Z 390.689,A -85,B 0,C 180,E1 -2963.649,E2 -2963.649} C_VEL
LIN {X 0,Y 558.869,Z 395.366,A -85,B 0,C 180,E1 -2964.588,E2 -2964.588} C_VEL
LIN {X 0,Y 558.869,Z 399.677,A -85,B 0,C 180,E1 -2965.673,E2 -2965.673} C_VEL
LIN {X 0,Y 558.836,Z 401.958,A -85,B 0,C 180,E1 -2966.395,E2 -2966.395} C_VEL
LIN {X 0,Y 558.799,Z 403.807,A -85,B 0,C 180,E1 -2967.116,E2 -2967.116} C_VEL
LIN {X 0,Y 558.745,Z 406.184,A -85,B 0,C 180,E1 -2968.558,E2 -2968.558} C_VEL
LIN {X 0,Y 558.74,Z 407,A -85,B 0,C 180,E1 -2970,E2 -2970} C_VEL
LIN {X 0,Y 558.745,Z 406.185,A -85,B 0,C 180,E1 -2971.441,E2 -2971.441} C_VEL
LIN {X 0,Y 558.799,Z 403.81,A -85,B 0,C 180,E1 -2972.883,E2 -2972.883} C_VEL
LIN {X 0,Y 558.844,Z 400.896,A -85,B 0,C 180,E1 -2973.966,E2 -2973.966} C_VEL
LIN {X 0,Y 558.798,Z 396.949,A -85,B 0,C 180,E1 -2975.051,E2 -2975.051} C_VEL
LIN {X 0,Y 558.922,Z 391.868,A -85,B 0,C 180,E1 -2976.135,E2 -2976.135} C_VEL
LIN {X 0,Y 558.978,Z 385.469,A -85,B 0,C 180,E1 -2977.223,E2 -2977.223} C_VEL
LIN {X 0,Y 559.099,Z 377.48,A -85,B 0,C 180,E1 -2978.311,E2 -2978.311} C_VEL
LIN {X 0,Y 559.195,Z 369.337,A -85,B 0,C 180,E1 -2979.221,E2 -2979.221} C_VEL
LIN {X 0,Y 559.362,Z 359.403,A -85,B 0,C 180,E1 -2980.131,E2 -2980.131} C_VEL
LIN {X 0,Y 559.505,Z 348.449,A -85,B 0,C 180,E1 -2980.934,E2 -2980.934} C_VEL
LIN {X 0,Y 559.636,Z 336.823,A -85,B 0,C 180,E1 -2981.61,E2 -2981.61} C_VEL
LIN {X 0,Y 559.814,Z 324.988,A -85,B 0,C 180,E1 -2982.138,E2 -2982.138} C_VEL
LIN {X 0,Y 559.958,Z 312.189,A -85,B 0,C 180,E1 -2982.549,E2 -2982.549} C_VEL
LIN {X 0,Y 559.765,Z 305.968,A -85,B 0,C 180,E1 -2982.7,E2 -2982.7} C_VEL
LIN {X 0,Y 558.925,Z 300.493,A -85,B 0,C 180,E1 -2982.827,E2 -2982.827} C_VEL
LIN {X 0,Y 558.968,Z 291.936,A -85,B 0,C 180,E1 -2985.683,E2 -2985.683} C_VEL
LIN {X 0,Y 559.02,Z 284.124,A -85,B 0,C 180,E1 -2988.318,E2 -2988.318} C_VEL
LIN {X 0,Y 559.09,Z 274.984,A -85,B 0,C 180,E1 -2991.379,E2 -2991.379} C_VEL
LIN {X 0,Y 559.131,Z 266.954,A -85,B 0,C 180,E1 -2994.111,E2 -2994.111} C_VEL
LIN {X 0,Y 559.15,Z 260.351,A -85,B 0,C 180,E1 -2996.462,E2 -2996.462} C_VEL
LIN {X 0,Y 559.276,Z 253.603,A -85,B 0,C 180,E1 -2998.933,E2 -2998.933} C_VEL
LIN {X 0,Y 559.378,Z 247.253,A -85,B 0,C 180,E1 -3001.311,E2 -3001.311} C_VEL
LIN {X 0,Y 559.501,Z 240.354,A -85,B 0,C 180,E1 -3003.999,E2 -3003.999} C_VEL
LIN {X 0,Y 559.549,Z 236.094,A -85,B 0,C 180,E1 -3005.735,E2 -3005.735} C_VEL
LIN {X 0,Y 559.193,Z 233.834,A -85,B 0,C 180,E1 -3006.752,E2 -3006.752} C_VEL
LIN {X 0,Y 559.178,Z 233.834,A -85,B 0,C 180,E1 -3009.865,E2 -3009.865} C_VEL
LIN {X 0,Y 559.163,Z 233.835,A -85,B 0,C 180,E1 -3012.742,E2 -3012.742} C_VEL
LIN {X 0,Y 559.151,Z 233.838,A -85,B 0,C 180,E1 -3015.76,E2 -3015.76} C_VEL
LIN {X 0,Y 559.189,Z 233.833,A -85,B 0,C 180,E1 -3018.231,E2 -3018.231} C_VEL
LIN {X 0,Y 559.175,Z 233.834,A -85,B 0,C 180,E1 -3021.19,E2 -3021.19} C_VEL
LIN {X 0,Y 559.17,Z 233.836,A -85,B 0,C 180,E1 -3023.791,E2 -3023.791} C_VEL
LIN {X 0,Y 559.161,Z 233.836,A -85,B 0,C 180,E1 -3026.424,E2 -3026.424} C_VEL
LIN {X 0,Y 559.163,Z 233.836,A -85,B 0,C 180,E1 -3028.981,E2 -3028.981} C_VEL
LIN {X 0,Y 559.165,Z 233.835,A -85,B 0,C 180,E1 -3031.617,E2 -3031.617} C_VEL
LIN {X 0,Y 559.177,Z 233.836,A -85,B 0,C 180,E1 -3033.902,E2 -3033.902} C_VEL
LIN {X 0,Y 559.151,Z 233.837,A -85,B 0,C 180,E1 -3036.566,E2 -3036.566} C_VEL
LIN {X 0,Y 559.174,Z 233.834,A -85,B 0,C 180,E1 -3039.395,E2 -3039.395} C_VEL
LIN {X 0,Y 559.15,Z 233.837,A -85,B 0,C 180,E1 -3041.685,E2 -3041.685} C_VEL
LIN {X 0,Y 559.165,Z 233.836,A -85,B 0,C 180,E1 -3043.947,E2 -3043.947} C_VEL
LIN {X 0,Y 559.169,Z 233.837,A -85,B 0,C 180,E1 -3046.183,E2 -3046.183} C_VEL
LIN {X 0,Y 559.204,Z 233.831,A -85,B 0,C 180,E1 -3049.133,E2 -3049.133} C_VEL
LIN {X 0,Y 559.204,Z 233.83,A -85,B 0,C 180,E1 -3052.053,E2 -3052.053} C_VEL
LIN {X 0,Y 559.253,Z 233.823,A -85,B 0,C 180,E1 -3054.953,E2 -3054.953} C_VEL
LIN {X 0,Y 559.243,Z 233.825,A -85,B 0,C 180,E1 -3057.839,E2 -3057.839} C_VEL
LIN {X 0,Y 559.269,Z 233.824,A -85,B 0,C 180,E1 -3060.719,E2 -3060.719} C_VEL
LIN {X 0,Y 559.237,Z 233.827,A -85,B 0,C 180,E1 -3062.881,E2 -3062.881} C_VEL
LIN {X 0,Y 559.223,Z 233.83,A -85,B 0,C 180,E1 -3065.769,E2 -3065.769} C_VEL
LIN {X 0,Y 559.197,Z 233.833,A -85,B 0,C 180,E1 -3068.673,E2 -3068.673} C_VEL
LIN {X 0,Y 559.133,Z 234.038,A -85,B 0,C 180,E1 -3070.867,E2 -3070.867} C_VEL
LIN {X 0,Y 559.094,Z 238.814,A -85,B 0,C 180,E1 -3073.817,E2 -3073.817} C_VEL
LIN {X 0,Y 559.046,Z 243.752,A -85,B 0,C 180,E1 -3076.806,E2 -3076.806} C_VEL
LIN {X 0,Y 558.982,Z 248.906,A -85,B 0,C 180,E1 -3079.843,E2 -3079.843} C_VEL
LIN {X 0,Y 558.944,Z 252.922,A -85,B 0,C 180,E1 -3082.16,E2 -3082.16} C_VEL
LIN {X 0,Y 558.879,Z 256.891,A -85,B 0,C 180,E1 -3084.517,E2 -3084.517} C_VEL
LIN {X 0,Y 558.831,Z 261.491,A -85,B 0,C 180,E1 -3087.186,E2 -3087.186} C_VEL
LIN {X 0,Y 558.783,Z 266.135,A -85,B 0,C 180,E1 -3089.794,E2 -3089.794} C_VEL
LIN {X 0,Y 558.78,Z 267.016,A -85,B 0,C 180,E1 -3090.272,E2 -3090.272} C_VEL
LIN {X 0,Y 558.082,Z 267.78,A -85,B 0,C 180,E1 -3090.665,E2 -3090.665} C_VEL
LIN {X 0,Y 552.344,Z 270.343,A -85,B 0,C 180,E1 -3091.898,E2 -3091.898} C_VEL
LIN {X 0,Y 551.673,Z 271.11,A -85,B 0,C 180,E1 -3092.299,E2 -3092.299} C_VEL
LIN {X 0,Y 551.705,Z 272.543,A -85,B 0,C 180,E1 -3093.077,E2 -3093.077} C_VEL
LIN {X 0,Y 553.027,Z 281.301,A -85,B 0,C 180,E1 -3093.313,E2 -3093.313} C_VEL
LIN {X 0,Y 552.865,Z 294.542,A -85,B 0,C 180,E1 -3093.734,E2 -3093.734} C_VEL
LIN {X 0,Y 552.695,Z 306.255,A -85,B 0,C 180,E1 -3094.258,E2 -3094.258} C_VEL
LIN {X 0,Y 552.533,Z 317.591,A -85,B 0,C 180,E1 -3094.915,E2 -3094.915} C_VEL
LIN {X 0,Y 552.345,Z 328.676,A -85,B 0,C 180,E1 -3095.724,E2 -3095.724} C_VEL
LIN {X 0,Y 552.16,Z 338.637,A -85,B 0,C 180,E1 -3096.633,E2 -3096.633} C_VEL
LIN {X 0,Y 552.025,Z 347.813,A -85,B 0,C 180,E1 -3097.668,E2 -3097.668} C_VEL
LIN {X 0,Y 551.906,Z 356.029,A -85,B 0,C 180,E1 -3098.816,E2 -3098.816} C_VEL
LIN {X 0,Y 551.843,Z 361.984,A -85,B 0,C 180,E1 -3099.854,E2 -3099.854} C_VEL
LIN {X 0,Y 551.744,Z 366.821,A -85,B 0,C 180,E1 -3100.897,E2 -3100.897} C_VEL
LIN {X 0,Y 551.746,Z 370.556,A -85,B 0,C 180,E1 -3101.921,E2 -3101.921} C_VEL
LIN {X 0,Y 551.667,Z 373.392,A -85,B 0,C 180,E1 -3102.949,E2 -3102.949} C_VEL
LIN {X 0,Y 551.69,Z 376.066,A -85,B 0,C 180,E1 -3104.477,E2 -3104.477} C_VEL
LIN {X 0,Y 551.69,Z 376.893,A -85,B 0,C 180,E1 -3105.522,E2 -3105.522} C_VEL
LIN {X 0,Y 551.656,Z 376.893,A -85,B 0,C 180,E1 -3106.564,E2 -3106.564} C_VEL
LIN {X 0,Y 551.645,Z 376.037,A -85,B 0,C 180,E1 -3107.638,E2 -3107.638} C_VEL
LIN {X 0,Y 551.676,Z 374.284,A -85,B 0,C 180,E1 -3108.729,E2 -3108.729} C_VEL
LIN {X 0,Y 551.716,Z 371.532,A -85,B 0,C 180,E1 -3109.843,E2 -3109.843} C_VEL
LIN {X 0,Y 551.766,Z 367.641,A -85,B 0,C 180,E1 -3110.982,E2 -3110.982} C_VEL
LIN {X 0,Y 551.809,Z 361.583,A -85,B 0,C 180,E1 -3112.314,E2 -3112.314} C_VEL
LIN {X 0,Y 551.929,Z 354.235,A -85,B 0,C 180,E1 -3113.545,E2 -3113.545} C_VEL
LIN {X 0,Y 552.025,Z 345.675,A -85,B 0,C 180,E1 -3114.687,E2 -3114.687} C_VEL
LIN {X 0,Y 552.21,Z 336.486,A -85,B 0,C 180,E1 -3115.669,E2 -3115.669} C_VEL
LIN {X 0,Y 552.378,Z 325.522,A -85,B 0,C 180,E1 -3116.615,E2 -3116.615} C_VEL
LIN {X 0,Y 552.532,Z 315.473,A -85,B 0,C 180,E1 -3117.313,E2 -3117.313} C_VEL
LIN {X 0,Y 552.663,Z 303.364,A -85,B 0,C 180,E1 -3117.977,E2 -3117.977} C_VEL
LIN {X 0,Y 552.923,Z 291.027,A -85,B 0,C 180,E1 -3118.483,E2 -3118.483} C_VEL
LIN {X 0,Y 552.84,Z 279.524,A -85,B 0,C 180,E1 -3118.827,E2 -3118.827} C_VEL
LIN {X 0,Y 551.685,Z 272.529,A -85,B 0,C 180,E1 -3119.021,E2 -3119.021} C_VEL
LIN {X 0,Y 551.681,Z 267.337,A -85,B 0,C 180,E1 -3121.879,E2 -3121.879} C_VEL
LIN {X 0,Y 551.748,Z 262.284,A -85,B 0,C 180,E1 -3124.736,E2 -3124.736} C_VEL
LIN {X 0,Y 551.799,Z 257.434,A -85,B 0,C 180,E1 -3127.537,E2 -3127.537} C_VEL
LIN {X 0,Y 551.881,Z 252.07,A -85,B 0,C 180,E1 -3130.665,E2 -3130.665} C_VEL
LIN {X 0,Y 551.899,Z 246.879,A -85,B 0,C 180,E1 -3133.731,E2 -3133.731} C_VEL
LIN {X 0,Y 551.967,Z 243.11,A -85,B 0,C 180,E1 -3136,E2 -3136} C_VEL
LIN {X 0,Y 552.075,Z 238.227,A -85,B 0,C 180,E1 -3138.992,E2 -3138.992} C_VEL
LIN {X 0,Y 552.033,Z 234.723,A -85,B 0,C 180,E1 -3141.213,E2 -3141.213} C_VEL
LIN {X 0,Y 552.127,Z 234.712,A -85,B 0,C 180,E1 -3143.422,E2 -3143.422} C_VEL
LIN {X 0,Y 552.221,Z 234.701,A -85,B 0,C 180,E1 -3144.889,E2 -3144.889} C_VEL
LIN {X 0,Y 552.211,Z 234.7,A -85,B 0,C 180,E1 -3147.812,E2 -3147.812} C_VEL
LIN {X 0,Y 552.237,Z 234.7,A -85,B 0,C 180,E1 -3150.729,E2 -3150.729} C_VEL
LIN {X 0,Y 552.2,Z 234.703,A -85,B 0,C 180,E1 -3152.918,E2 -3152.918} C_VEL
LIN {X 0,Y 552.19,Z 234.704,A -85,B 0,C 180,E1 -3155.844,E2 -3155.844} C_VEL
LIN {X 0,Y 552.163,Z 234.707,A -85,B 0,C 180,E1 -3158.786,E2 -3158.786} C_VEL
LIN {X 0,Y 552.154,Z 234.71,A -85,B 0,C 180,E1 -3161.751,E2 -3161.751} C_VEL
LIN {X 0,Y 552.126,Z 234.711,A -85,B 0,C 180,E1 -3164.748,E2 -3164.748} C_VEL
LIN {X 0,Y 552.105,Z 234.716,A -85,B 0,C 180,E1 -3167.788,E2 -3167.788} C_VEL
LIN {X 0,Y 552.124,Z 234.714,A -85,B 0,C 180,E1 -3170.101,E2 -3170.101} C_VEL
LIN {X 0,Y 552.104,Z 234.716,A -85,B 0,C 180,E1 -3172.45,E2 -3172.45} C_VEL
LIN {X 0,Y 552.145,Z 234.708,A -85,B 0,C 180,E1 -3175.351,E2 -3175.351} C_VEL
LIN {X 0,Y 552.117,Z 234.713,A -85,B 0,C 180,E1 -3178.097,E2 -3178.097} C_VEL
LIN {X 0,Y 552.104,Z 234.715,A -85,B 0,C 180,E1 -3180.609,E2 -3180.609} C_VEL
LIN {X 0,Y 552.112,Z 234.715,A -85,B 0,C 180,E1 -3183.185,E2 -3183.185} C_VEL
LIN {X 0,Y 552.102,Z 234.715,A -85,B 0,C 180,E1 -3185.842,E2 -3185.842} C_VEL
LIN {X 0,Y 552.116,Z 234.713,A -85,B 0,C 180,E1 -3189.062,E2 -3189.062} C_VEL
LIN {X 0,Y 552.13,Z 234.712,A -85,B 0,C 180,E1 -3191.444,E2 -3191.444} C_VEL
LIN {X 0,Y 552.085,Z 234.715,A -85,B 0,C 180,E1 -3194.532,E2 -3194.532} C_VEL
LIN {X 0,Y 552.121,Z 234.715,A -85,B 0,C 180,E1 -3197.585,E2 -3197.585} C_VEL
LIN {X 0,Y 552.124,Z 234.711,A -85,B 0,C 180,E1 -3200.474,E2 -3200.474} C_VEL
LIN {X 0,Y 552.111,Z 234.714,A -85,B 0,C 180,E1 -3203.315,E2 -3203.315} C_VEL
LIN {X 0,Y 552.12,Z 234.714,A -85,B 0,C 180,E1 -3205.94,E2 -3205.94} C_VEL
LIN {X 0,Y 552.107,Z 234.716,A -85,B 0,C 180,E1 -3208.541,E2 -3208.541} C_VEL
LIN {X 0,Y 552.115,Z 234.712,A -85,B 0,C 180,E1 -3211.438,E2 -3211.438} C_VEL
LIN {X 0,Y 552.128,Z 234.712,A -85,B 0,C 180,E1 -3214.357,E2 -3214.357} C_VEL
LIN {X 0,Y 552.101,Z 234.717,A -85,B 0,C 180,E1 -3216.759,E2 -3216.759} C_VEL
LIN {X 0,Y 552.118,Z 234.715,A -85,B 0,C 180,E1 -3219.121,E2 -3219.121} C_VEL
LIN {X 0,Y 552.122,Z 234.713,A -85,B 0,C 180,E1 -3221.445,E2 -3221.445} C_VEL
LIN {X 0,Y 552.112,Z 234.713,A -85,B 0,C 180,E1 -3223.738,E2 -3223.738} C_VEL
LIN {X 0,Y 552.127,Z 234.71,A -85,B 0,C 180,E1 -3226.005,E2 -3226.005} C_VEL
LIN {X 0,Y 552.171,Z 234.706,A -85,B 0,C 180,E1 -3228.995,E2 -3228.995} C_VEL
LIN {X 0,Y 552.156,Z 234.707,A -85,B 0,C 180,E1 -3231.952,E2 -3231.952} C_VEL
LIN {X 0,Y 552.224,Z 234.701,A -85,B 0,C 180,E1 -3234.89,E2 -3234.89} C_VEL
LIN {X 0,Y 552.218,Z 234.699,A -85,B 0,C 180,E1 -3237.813,E2 -3237.813} C_VEL
LIN {X 0,Y 552.24,Z 234.699,A -85,B 0,C 180,E1 -3240.73,E2 -3240.73} C_VEL
LIN {X 0,Y 552.199,Z 234.703,A -85,B 0,C 180,E1 -3242.919,E2 -3242.919} C_VEL
LIN {X 0,Y 552.192,Z 234.704,A -85,B 0,C 180,E1 -3245.845,E2 -3245.845} C_VEL
LIN {X 0,Y 552.153,Z 234.707,A -85,B 0,C 180,E1 -3248.787,E2 -3248.787} C_VEL
LIN {X 0,Y 552.157,Z 234.709,A -85,B 0,C 180,E1 -3251.751,E2 -3251.751} C_VEL
LIN {X 0,Y 552.131,Z 234.71,A -85,B 0,C 180,E1 -3254.749,E2 -3254.749} C_VEL
LIN {X 0,Y 552.106,Z 234.715,A -85,B 0,C 180,E1 -3257.789,E2 -3257.789} C_VEL
LIN {X 0,Y 552.126,Z 234.713,A -85,B 0,C 180,E1 -3260.102,E2 -3260.102} C_VEL
LIN {X 0,Y 552.092,Z 234.717,A -85,B 0,C 180,E1 -3262.452,E2 -3262.452} C_VEL
LIN {X 0,Y 552.152,Z 234.708,A -85,B 0,C 180,E1 -3265.351,E2 -3265.351} C_VEL
LIN {X 0,Y 552.123,Z 234.712,A -85,B 0,C 180,E1 -3268.098,E2 -3268.098} C_VEL
LIN {X 0,Y 552.101,Z 234.715,A -85,B 0,C 180,E1 -3270.61,E2 -3270.61} C_VEL
LIN {X 0,Y 552.105,Z 234.716,A -85,B 0,C 180,E1 -3273.187,E2 -3273.187} C_VEL
LIN {X 0,Y 552.101,Z 234.715,A -85,B 0,C 180,E1 -3275.843,E2 -3275.843} C_VEL
LIN {X 0,Y 552.124,Z 234.713,A -85,B 0,C 180,E1 -3279.063,E2 -3279.063} C_VEL
LIN {X 0,Y 552.127,Z 234.713,A -85,B 0,C 180,E1 -3281.446,E2 -3281.446} C_VEL
LIN {X 0,Y 552.092,Z 234.715,A -85,B 0,C 180,E1 -3284.532,E2 -3284.532} C_VEL
LIN {X 0,Y 552.131,Z 234.713,A -85,B 0,C 180,E1 -3287.585,E2 -3287.585} C_VEL
LIN {X 0,Y 552.132,Z 234.71,A -85,B 0,C 180,E1 -3290.474,E2 -3290.474} C_VEL
LIN {X 0,Y 552.134,Z 234.719,A -85,B 0,C 180,E1 -3293.142,E2 -3293.142} C_VEL
LIN {X 0,Y 552.544,Z 237.917,A -85,B 0,C 180,E1 -3294.493,E2 -3294.493} C_VEL
LIN {X 0,Y 552.489,Z 244.405,A -85,B 0,C 180,E1 -3297.095,E2 -3297.095} C_VEL
LIN {X 0,Y 552.33,Z 251.692,A -85,B 0,C 180,E1 -3299.912,E2 -3299.912} C_VEL
LIN {X 0,Y 552.169,Z 259.168,A -85,B 0,C 180,E1 -3302.729,E2 -3302.729} C_VEL
LIN {X 0,Y 552.084,Z 267.027,A -85,B 0,C 180,E1 -3305.561,E2 -3305.561} C_VEL
LIN {X 0,Y 552.047,Z 274.969,A -85,B 0,C 180,E1 -3308.334,E2 -3308.334} C_VEL
LIN {X 0,Y 551.983,Z 282.892,A -85,B 0,C 180,E1 -3311.055,E2 -3311.055} C_VEL
LIN {X 0,Y 551.905,Z 291.923,A -85,B 0,C 180,E1 -3314.111,E2 -3314.111} C_VEL
LIN {X 0,Y 551.84,Z 300.492,A -85,B 0,C 180,E1 -3317.005,E2 -3317.005} C_VEL
LIN {X 0,Y 553.089,Z 309.441,A -85,B 0,C 180,E1 -3317.222,E2 -3317.222} C_VEL
LIN {X 0,Y 552.917,Z 322.478,A -85,B 0,C 180,E1 -3317.614,E2 -3317.614} C_VEL
LIN {X 0,Y 552.743,Z 333.493,A -85,B 0,C 180,E1 -3318.076,E2 -3318.076} C_VEL
LIN {X 0,Y 552.57,Z 345.199,A -85,B 0,C 180,E1 -3318.715,E2 -3318.715} C_VEL
LIN {X 0,Y 552.426,Z 357.095,A -85,B 0,C 180,E1 -3319.555,E2 -3319.555} C_VEL
LIN {X 0,Y 552.202,Z 367.54,A -85,B 0,C 180,E1 -3320.476,E2 -3320.476} C_VEL
LIN {X 0,Y 552.082,Z 375.992,A -85,B 0,C 180,E1 -3321.398,E2 -3321.398} C_VEL
LIN {X 0,Y 551.927,Z 384.236,A -85,B 0,C 180,E1 -3322.5,E2 -3322.5} C_VEL
LIN {X 0,Y 551.822,Z 391.21,A -85,B 0,C 180,E1 -3323.663,E2 -3323.663} C_VEL
LIN {X 0,Y 551.724,Z 396.95,A -85,B 0,C 180,E1 -3324.884,E2 -3324.884} C_VEL
LIN {X 0,Y 551.764,Z 400.894,A -85,B 0,C 180,E1 -3325.983,E2 -3325.983} C_VEL
LIN {X 0,Y 551.724,Z 403.807,A -85,B 0,C 180,E1 -3327.079,E2 -3327.079} C_VEL
LIN {X 0,Y 551.645,Z 406.183,A -85,B 0,C 180,E1 -3328.54,E2 -3328.54} C_VEL
LIN {X 0,Y 551.64,Z 407,A -85,B 0,C 180,E1 -3330,E2 -3330} C_VEL
LIN {X 0,Y 551.645,Z 406.185,A -85,B 0,C 180,E1 -3331.46,E2 -3331.46} C_VEL
LIN {X 0,Y 551.724,Z 403.81,A -85,B 0,C 180,E1 -3332.92,E2 -3332.92} C_VEL
LIN {X 0,Y 551.764,Z 400.896,A -85,B 0,C 180,E1 -3334.017,E2 -3334.017} C_VEL
LIN {X 0,Y 551.724,Z 396.949,A -85,B 0,C 180,E1 -3335.116,E2 -3335.116} C_VEL
LIN {X 0,Y 551.816,Z 391.126,A -85,B 0,C 180,E1 -3336.353,E2 -3336.353} C_VEL
LIN {X 0,Y 551.927,Z 384.238,A -85,B 0,C 180,E1 -3337.499,E2 -3337.499} C_VEL
LIN {X 0,Y 552.082,Z 375.994,A -85,B 0,C 180,E1 -3338.602,E2 -3338.602} C_VEL
LIN {X 0,Y 552.201,Z 367.542,A -85,B 0,C 180,E1 -3339.523,E2 -3339.523} C_VEL
LIN {X 0,Y 552.426,Z 357.097,A -85,B 0,C 180,E1 -3340.445,E2 -3340.445} C_VEL
LIN {X 0,Y 552.579,Z 345.351,A -85,B 0,C 180,E1 -3341.275,E2 -3341.275} C_VEL
LIN {X 0,Y 552.741,Z 333.495,A -85,B 0,C 180,E1 -3341.924,E2 -3341.924} C_VEL
LIN {X 0,Y 552.958,Z 321.175,A -85,B 0,C 180,E1 -3342.431,E2 -3342.431} C_VEL
LIN {X 0,Y 553.06,Z 308.049,A -85,B 0,C 180,E1 -3342.814,E2 -3342.814} C_VEL
LIN {X 0,Y 551.84,Z 300.493,A -85,B 0,C 180,E1 -3342.994,E2 -3342.994} C_VEL
LIN {X 0,Y 551.905,Z 291.918,A -85,B 0,C 180,E1 -3345.889,E2 -3345.889} C_VEL
LIN {X 0,Y 551.966,Z 282.809,A -85,B 0,C 180,E1 -3348.946,E2 -3348.946} C_VEL
LIN {X 0,Y 552.041,Z 273.662,A -85,B 0,C 180,E1 -3352.059,E2 -3352.059} C_VEL
LIN {X 0,Y 552.073,Z 265.717,A -85,B 0,C 180,E1 -3354.84,E2 -3354.84} C_VEL
LIN {X 0,Y 552.199,Z 257.97,A -85,B 0,C 180,E1 -3357.68,E2 -3357.68} C_VEL
LIN {X 0,Y 552.382,Z 250.195,A -85,B 0,C 180,E1 -3360.591,E2 -3360.591} C_VEL
LIN {X 0,Y 552.495,Z 242.544,A -85,B 0,C 180,E1 -3363.596,E2 -3363.596} C_VEL
LIN {X 0,Y 552.544,Z 237.169,A -85,B 0,C 180,E1 -3365.808,E2 -3365.808} C_VEL
LIN {X 0,Y 552.143,Z 234.712,A -85,B 0,C 180,E1 -3366.971,E2 -3366.971} C_VEL
LIN {X 0,Y 552.128,Z 234.713,A -85,B 0,C 180,E1 -3369.526,E2 -3369.526} C_VEL
LIN {X 0,Y 552.13,Z 234.713,A -85,B 0,C 180,E1 -3372.424,E2 -3372.424} C_VEL
LIN {X 0,Y 552.096,Z 234.718,A -85,B 0,C 180,E1 -3375.562,E2 -3375.562} C_VEL
LIN {X 0,Y 552.138,Z 234.712,A -85,B 0,C 180,E1 -3378.675,E2 -3378.675} C_VEL
LIN {X 0,Y 552.117,Z 234.714,A -85,B 0,C 180,E1 -3381.41,E2 -3381.41} C_VEL
LIN {X 0,Y 552.11,Z 234.714,A -85,B 0,C 180,E1 -3384.158,E2 -3384.158} C_VEL
LIN {X 0,Y 552.119,Z 234.714,A -85,B 0,C 180,E1 -3386.814,E2 -3386.814} C_VEL
LIN {X 0,Y 552.11,Z 234.714,A -85,B 0,C 180,E1 -3389.391,E2 -3389.391} C_VEL
LIN {X 0,Y 552.121,Z 234.714,A -85,B 0,C 180,E1 -3391.902,E2 -3391.902} C_VEL
LIN {X 0,Y 552.15,Z 234.709,A -85,B 0,C 180,E1 -3394.649,E2 -3394.649} C_VEL
LIN {X 0,Y 552.09,Z 234.716,A -85,B 0,C 180,E1 -3397.548,E2 -3397.548} C_VEL
LIN {X 0,Y 552.151,Z 234.709,A -85,B 0,C 180,E1 -3400.674,E2 -3400.674} C_VEL
LIN {X 0,Y 552.115,Z 234.713,A -85,B 0,C 180,E1 -3403.736,E2 -3403.736} C_VEL
LIN {X 0,Y 552.132,Z 234.712,A -85,B 0,C 180,E1 -3406.004,E2 -3406.004} C_VEL
LIN {X 0,Y 552.172,Z 234.706,A -85,B 0,C 180,E1 -3408.993,E2 -3408.993} C_VEL
LIN {X 0,Y 552.158,Z 234.708,A -85,B 0,C 180,E1 -3411.951,E2 -3411.951} C_VEL
LIN {X 0,Y 552.227,Z 234.699,A -85,B 0,C 180,E1 -3414.888,E2 -3414.888} C_VEL
LIN {X 0,Y 552.215,Z 234.701,A -85,B 0,C 180,E1 -3417.811,E2 -3417.811} C_VEL
LIN {X 0,Y 552.238,Z 234.699,A -85,B 0,C 180,E1 -3420.728,E2 -3420.728} C_VEL
LIN {X 0,Y 552.203,Z 234.703,A -85,B 0,C 180,E1 -3422.917,E2 -3422.917} C_VEL
LIN {X 0,Y 552.194,Z 234.705,A -85,B 0,C 180,E1 -3425.843,E2 -3425.843} C_VEL
LIN {X 0,Y 552.164,Z 234.71,A -85,B 0,C 180,E1 -3428.785,E2 -3428.785} C_VEL
LIN {X 0,Y 552.078,Z 234.72,A -85,B 0,C 180,E1 -3430.265,E2 -3430.265} C_VEL
LIN {X 0,Y 552.106,Z 235.153,A -85,B 0,C 180,E1 -3431.007,E2 -3431.007} C_VEL
LIN {X 0,Y 552.041,Z 239.934,A -85,B 0,C 180,E1 -3433.997,E2 -3433.997} C_VEL
LIN {X 0,Y 551.98,Z 244.889,A -85,B 0,C 180,E1 -3437.027,E2 -3437.027} C_VEL
LIN {X 0,Y 551.912,Z 250.047,A -85,B 0,C 180,E1 -3440.108,E2 -3440.108} C_VEL
LIN {X 0,Y 551.887,Z 254.114,A -85,B 0,C 180,E1 -3442.459,E2 -3442.459} C_VEL
LIN {X 0,Y 551.82,Z 258.84,A -85,B 0,C 180,E1 -3445.279,E2 -3445.279} C_VEL
LIN {X 0,Y 551.778,Z 263.701,A -85,B 0,C 180,E1 -3448.115,E2 -3448.115} C_VEL
LIN {X 0,Y 551.716,Z 269.488,A -85,B 0,C 180,E1 -3451.41,E2 -3451.41} C_VEL
LIN {X 0,Y 551.673,Z 271.11,A -85,B 0,C 180,E1 -3452.299,E2 -3452.299} C_VEL
LIN {X 0,Y 551.512,Z 272.28,A -85,B 0,C 180,E1 -3452.579,E2 -3452.579} C_VEL
LIN {X 0,Y 550.943,Z 275.072,A -85,B 0,C 180,E1 -3452.871,E2 -3452.871} C_VEL
LIN {X 0,Y 549.87,Z 279.652,A -85,B 0,C 180,E1 -3453.128,E2 -3453.128} C_VEL
LIN {X 0,Y 548.305,Z 285.515,A -85,B 0,C 180,E1 -3453.32,E2 -3453.32} C_VEL
LIN {X 0,Y 546.247,Z 292.212,A -85,B 0,C 180,E1 -3453.494,E2 -3453.494} C_VEL
LIN {X 0,Y 545.86,Z 298.89,A -85,B 0,C 180,E1 -3453.754,E2 -3453.754} C_VEL
LIN {X 0,Y 545.67,Z 309.837,A -85,B 0,C 180,E1 -3454.295,E2 -3454.295} C_VEL
LIN {X 0,Y 545.502,Z 320.685,A -85,B 0,C 180,E1 -3454.98,E2 -3454.98} C_VEL
LIN {X 0,Y 545.293,Z 331.246,A -85,B 0,C 180,E1 -3455.812,E2 -3455.812} C_VEL
LIN {X 0,Y 545.112,Z 341.188,A -85,B 0,C 180,E1 -3456.779,E2 -3456.779} C_VEL
LIN {X 0,Y 544.951,Z 349.017,A -85,B 0,C 180,E1 -3457.71,E2 -3457.71} C_VEL
LIN {X 0,Y 544.833,Z 356.058,A -85,B 0,C 180,E1 -3458.726,E2 -3458.726} C_VEL
LIN {X 0,Y 544.745,Z 362.771,A -85,B 0,C 180,E1 -3459.934,E2 -3459.934} C_VEL
LIN {X 0,Y 544.666,Z 368.054,A -85,B 0,C 180,E1 -3461.151,E2 -3461.151} C_VEL
LIN {X 0,Y 544.648,Z 371.375,A -85,B 0,C 180,E1 -3462.142,E2 -3462.142} C_VEL
LIN {X 0,Y 544.573,Z 373.951,A -85,B 0,C 180,E1 -3463.155,E2 -3463.155} C_VEL
LIN {X 0,Y 544.569,Z 375.728,A -85,B 0,C 180,E1 -3464.177,E2 -3464.177} C_VEL
LIN {X 0,Y 544.575,Z 376.729,A -85,B 0,C 180,E1 -3465.217,E2 -3465.217} C_VEL
LIN {X 0,Y 544.563,Z 376.956,A -85,B 0,C 180,E1 -3466.278,E2 -3466.278} C_VEL
LIN {X 0,Y 544.535,Z 376.358,A -85,B 0,C 180,E1 -3467.362,E2 -3467.362} C_VEL
LIN {X 0,Y 544.593,Z 374.881,A -85,B 0,C 180,E1 -3468.458,E2 -3468.458} C_VEL
LIN {X 0,Y 544.638,Z 371.739,A -85,B 0,C 180,E1 -3469.82,E2 -3469.82} C_VEL
LIN {X 0,Y 544.661,Z 368.652,A -85,B 0,C 180,E1 -3470.783,E2 -3470.783} C_VEL
LIN {X 0,Y 544.717,Z 363.986,A -85,B 0,C 180,E1 -3471.907,E2 -3471.907} C_VEL
LIN {X 0,Y 544.795,Z 357.582,A -85,B 0,C 180,E1 -3473.11,E2 -3473.11} C_VEL
LIN {X 0,Y 544.912,Z 350.354,A -85,B 0,C 180,E1 -3474.198,E2 -3474.198} C_VEL
LIN {X 0,Y 545.067,Z 342.095,A -85,B 0,C 180,E1 -3475.212,E2 -3475.212} C_VEL
LIN {X 0,Y 545.25,Z 333.057,A -85,B 0,C 180,E1 -3476.12,E2 -3476.12} C_VEL
LIN {X 0,Y 545.408,Z 322.702,A -85,B 0,C 180,E1 -3476.964,E2 -3476.964} C_VEL
LIN {X 0,Y 545.57,Z 311.745,A -85,B 0,C 180,E1 -3477.684,E2 -3477.684} C_VEL
LIN {X 0,Y 545.801,Z 300.381,A -85,B 0,C 180,E1 -3478.271,E2 -3478.271} C_VEL
LIN {X 0,Y 546.02,Z 287.691,A -85,B 0,C 180,E1 -3478.757,E2 -3478.757} C_VEL
LIN {X 0,Y 545.887,Z 280.12,A -85,B 0,C 180,E1 -3478.978,E2 -3478.978} C_VEL
LIN {X 0,Y 544.581,Z 272.59,A -85,B 0,C 180,E1 -3479.192,E2 -3479.192} C_VEL
LIN {X 0,Y 544.602,Z 267.046,A -85,B 0,C 180,E1 -3482.318,E2 -3482.318} C_VEL
LIN {X 0,Y 544.666,Z 262.722,A -85,B 0,C 180,E1 -3484.799,E2 -3484.799} C_VEL
LIN {X 0,Y 544.706,Z 258.576,A -85,B 0,C 180,E1 -3487.228,E2 -3487.228} C_VEL
LIN {X 0,Y 544.832,Z 253.297,A -85,B 0,C 180,E1 -3490.327,E2 -3490.327} C_VEL
LIN {X 0,Y 544.832,Z 247.975,A -85,B 0,C 180,E1 -3493.514,E2 -3493.514} C_VEL
LIN {X 0,Y 544.929,Z 244.19,A -85,B 0,C 180,E1 -3495.816,E2 -3495.816} C_VEL
LIN {X 0,Y 545.026,Z 239.271,A -85,B 0,C 180,E1 -3498.848,E2 -3498.848} C_VEL
LIN {X 0,Y 544.987,Z 235.702,A -85,B 0,C 180,E1 -3501.098,E2 -3501.098} C_VEL
LIN {X 0,Y 545.11,Z 235.586,A -85,B 0,C 180,E1 -3503.337,E2 -3503.337} C_VEL
LIN {X 0,Y 545.196,Z 235.577,A -85,B 0,C 180,E1 -3504.823,E2 -3504.823} C_VEL
LIN {X 0,Y 545.183,Z 235.575,A -85,B 0,C 180,E1 -3507.784,E2 -3507.784} C_VEL
LIN {X 0,Y 545.206,Z 235.576,A -85,B 0,C 180,E1 -3510.739,E2 -3510.739} C_VEL
LIN {X 0,Y 545.166,Z 235.579,A -85,B 0,C 180,E1 -3512.956,E2 -3512.956} C_VEL
LIN {X 0,Y 545.161,Z 235.579,A -85,B 0,C 180,E1 -3515.92,E2 -3515.92} C_VEL
LIN {X 0,Y 545.12,Z 235.584,A -85,B 0,C 180,E1 -3518.9,E2 -3518.9} C_VEL
LIN {X 0,Y 545.125,Z 235.584,A -85,B 0,C 180,E1 -3521.904,E2 -3521.904} C_VEL
LIN {X 0,Y 545.075,Z 235.59,A -85,B 0,C 180,E1 -3524.944,E2 -3524.944} C_VEL
LIN {X 0,Y 545.073,Z 235.59,A -85,B 0,C 180,E1 -3528.026,E2 -3528.026} C_VEL
LIN {X 0,Y 545.089,Z 235.588,A -85,B 0,C 180,E1 -3530.372,E2 -3530.372} C_VEL
LIN {X 0,Y 545.104,Z 235.588,A -85,B 0,C 180,E1 -3533.558,E2 -3533.558} C_VEL
LIN {X 0,Y 545.078,Z 235.592,A -85,B 0,C 180,E1 -3536,E2 -3536} C_VEL
LIN {X 0,Y 545.083,Z 235.588,A -85,B 0,C 180,E1 -3538.75,E2 -3538.75} C_VEL
LIN {X 0,Y 545.067,Z 235.591,A -85,B 0,C 180,E1 -3541.683,E2 -3541.683} C_VEL
LIN {X 0,Y 545.07,Z 235.591,A -85,B 0,C 180,E1 -3544.563,E2 -3544.563} C_VEL
LIN {X 0,Y 545.029,Z 235.595,A -85,B 0,C 180,E1 -3547.304,E2 -3547.304} C_VEL
LIN {X 0,Y 545.082,Z 235.589,A -85,B 0,C 180,E1 -3550.14,E2 -3550.14} C_VEL
LIN {X 0,Y 545.077,Z 235.59,A -85,B 0,C 180,E1 -3553.106,E2 -3553.106} C_VEL
LIN {X 0,Y 545.055,Z 235.593,A -85,B 0,C 180,E1 -3556.225,E2 -3556.225} C_VEL
LIN {X 0,Y 545.091,Z 235.59,A -85,B 0,C 180,E1 -3558.888,E2 -3558.888} C_VEL
LIN {X 0,Y 545.043,Z 235.593,A -85,B 0,C 180,E1 -3561.763,E2 -3561.763} C_VEL
LIN {X 0,Y 545.054,Z 235.592,A -85,B 0,C 180,E1 -3564.534,E2 -3564.534} C_VEL
LIN {X 0,Y 545.071,Z 235.593,A -85,B 0,C 180,E1 -3567.213,E2 -3567.213} C_VEL
LIN {X 0,Y 545.091,Z 235.588,A -85,B 0,C 180,E1 -3569.813,E2 -3569.813} C_VEL
LIN {X 0,Y 545.091,Z 235.588,A -85,B 0,C 180,E1 -3572.825,E2 -3572.825} C_VEL
LIN {X 0,Y 545.043,Z 235.595,A -85,B 0,C 180,E1 -3575.632,E2 -3575.632} C_VEL
LIN {X 0,Y 545.06,Z 235.592,A -85,B 0,C 180,E1 -3578.838,E2 -3578.838} C_VEL
LIN {X 0,Y 545.075,Z 235.59,A -85,B 0,C 180,E1 -3581.197,E2 -3581.197} C_VEL
LIN {X 0,Y 545.068,Z 235.59,A -85,B 0,C 180,E1 -3583.522,E2 -3583.522} C_VEL
LIN {X 0,Y 545.086,Z 235.587,A -85,B 0,C 180,E1 -3585.821,E2 -3585.821} C_VEL
LIN {X 0,Y 545.125,Z 235.585,A -85,B 0,C 180,E1 -3588.851,E2 -3588.851} C_VEL
LIN {X 0,Y 545.126,Z 235.582,A -85,B 0,C 180,E1 -3591.848,E2 -3591.848} C_VEL
LIN {X 0,Y 545.199,Z 235.576,A -85,B 0,C 180,E1 -3594.824,E2 -3594.824} C_VEL
LIN {X 0,Y 545.189,Z 235.575,A -85,B 0,C 180,E1 -3597.785,E2 -3597.785} C_VEL
LIN {X 0,Y 545.21,Z 235.575,A -85,B 0,C 180,E1 -3600.739,E2 -3600.739} C_VEL
LIN {X 0,Y 545.166,Z 235.579,A -85,B 0,C 180,E1 -3602.957,E2 -3602.957} C_VEL
LIN {X 0,Y 545.164,Z 235.579,A -85,B 0,C 180,E1 -3605.92,E2 -3605.92} C_VEL
LIN {X 0,Y 545.112,Z 235.585,A -85,B 0,C 180,E1 -3608.901,E2 -3608.901} C_VEL
LIN {X 0,Y 545.13,Z 235.583,A -85,B 0,C 180,E1 -3611.905,E2 -3611.905} C_VEL
LIN {X 0,Y 545.08,Z 235.589,A -85,B 0,C 180,E1 -3614.944,E2 -3614.944} C_VEL
LIN {X 0,Y 545.074,Z 235.59,A -85,B 0,C 180,E1 -3618.027,E2 -3618.027} C_VEL
LIN {X 0,Y 545.091,Z 235.587,A -85,B 0,C 180,E1 -3620.373,E2 -3620.373} C_VEL
LIN {X 0,Y 545.087,Z 235.59,A -85,B 0,C 180,E1 -3623.56,E2 -3623.56} C_VEL
LIN {X 0,Y 545.076,Z 235.592,A -85,B 0,C 180,E1 -3626.001,E2 -3626.001} C_VEL
LIN {X 0,Y 545.087,Z 235.588,A -85,B 0,C 180,E1 -3628.749,E2 -3628.749} C_VEL
LIN {X 0,Y 545.055,Z 235.593,A -85,B 0,C 180,E1 -3631.68,E2 -3631.68} C_VEL
LIN {X 0,Y 545.075,Z 235.592,A -85,B 0,C 180,E1 -3634.564,E2 -3634.564} C_VEL
LIN {X 0,Y 545.036,Z 235.594,A -85,B 0,C 180,E1 -3637.305,E2 -3637.305} C_VEL
LIN {X 0,Y 545.07,Z 235.59,A -85,B 0,C 180,E1 -3640.143,E2 -3640.143} C_VEL
LIN {X 0,Y 545.077,Z 235.59,A -85,B 0,C 180,E1 -3643.107,E2 -3643.107} C_VEL
LIN {X 0,Y 545.048,Z 235.593,A -85,B 0,C 180,E1 -3646.227,E2 -3646.227} C_VEL
LIN {X 0,Y 545.096,Z 235.589,A -85,B 0,C 180,E1 -3648.888,E2 -3648.888} C_VEL
LIN {X 0,Y 545.052,Z 235.592,A -85,B 0,C 180,E1 -3651.763,E2 -3651.763} C_VEL
LIN {X 0,Y 545.097,Z 235.6,A -85,B 0,C 180,E1 -3652.974,E2 -3652.974} C_VEL
LIN {X 0,Y 545.564,Z 239.339,A -85,B 0,C 180,E1 -3654.572,E2 -3654.572} C_VEL
LIN {X 0,Y 545.458,Z 245.914,A -85,B 0,C 180,E1 -3657.238,E2 -3657.238} C_VEL
LIN {X 0,Y 545.306,Z 253.639,A -85,B 0,C 180,E1 -3660.252,E2 -3660.252} C_VEL
LIN {X 0,Y 545.101,Z 261.334,A -85,B 0,C 180,E1 -3663.176,E2 -3663.176} C_VEL
LIN {X 0,Y 545.042,Z 268.051,A -85,B 0,C 180,E1 -3665.631,E2 -3665.631} C_VEL
LIN {X 0,Y 544.98,Z 275.328,A -85,B 0,C 180,E1 -3668.204,E2 -3668.204} C_VEL
LIN {X 0,Y 544.89,Z 283.913,A -85,B 0,C 180,E1 -3671.189,E2 -3671.189} C_VEL
LIN {X 0,Y 544.847,Z 292.944,A -85,B 0,C 180,E1 -3674.284,E2 -3674.284} C_VEL
LIN {X 0,Y 544.759,Z 300.474,A -85,B 0,C 180,E1 -3676.833,E2 -3676.833} C_VEL
LIN {X 0,Y 546.168,Z 310.356,A -85,B 0,C 180,E1 -3677.081,E2 -3677.081} C_VEL
LIN {X 0,Y 545.98,Z 322.478,A -85,B 0,C 180,E1 -3677.454,E2 -3677.454} C_VEL
LIN {X 0,Y 545.785,Z 333.491,A -85,B 0,C 180,E1 -3677.922,E2 -3677.922} C_VEL
LIN {X 0,Y 545.592,Z 345.598,A -85,B 0,C 180,E1 -3678.595,E2 -3678.595} C_VEL
LIN {X 0,Y 545.422,Z 357.093,A -85,B 0,C 180,E1 -3679.42,E2 -3679.42} C_VEL
LIN {X 0,Y 545.166,Z 367.54,A -85,B 0,C 180,E1 -3680.352,E2 -3680.352} C_VEL
LIN {X 0,Y 545.029,Z 375.992,A -85,B 0,C 180,E1 -3681.285,E2 -3681.285} C_VEL
LIN {X 0,Y 544.86,Z 384.235,A -85,B 0,C 180,E1 -3682.403,E2 -3682.403} C_VEL
LIN {X 0,Y 544.734,Z 391.619,A -85,B 0,C 180,E1 -3683.656,E2 -3683.656} C_VEL
LIN {X 0,Y 544.654,Z 396.95,A -85,B 0,C 180,E1 -3684.818,E2 -3684.818} C_VEL
LIN {X 0,Y 544.684,Z 400.894,A -85,B 0,C 180,E1 -3685.931,E2 -3685.931} C_VEL
LIN {X 0,Y 544.651,Z 403.807,A -85,B 0,C 180,E1 -3687.041,E2 -3687.041} C_VEL
LIN {X 0,Y 544.546,Z 406.182,A -85,B 0,C 180,E1 -3688.521,E2 -3688.521} C_VEL
LIN {X 0,Y 544.541,Z 407,A -85,B 0,C 180,E1 -3690,E2 -3690} C_VEL
LIN {X 0,Y 544.546,Z 406.184,A -85,B 0,C 180,E1 -3691.479,E2 -3691.479} C_VEL
LIN {X 0,Y 544.651,Z 403.81,A -85,B 0,C 180,E1 -3692.958,E2 -3692.958} C_VEL
LIN {X 0,Y 544.684,Z 400.896,A -85,B 0,C 180,E1 -3694.069,E2 -3694.069} C_VEL
LIN {X 0,Y 544.654,Z 396.949,A -85,B 0,C 180,E1 -3695.182,E2 -3695.182} C_VEL
LIN {X 0,Y 544.73,Z 391.646,A -85,B 0,C 180,E1 -3696.339,E2 -3696.339} C_VEL
LIN {X 0,Y 544.86,Z 384.237,A -85,B 0,C 180,E1 -3697.597,E2 -3697.597} C_VEL
LIN {X 0,Y 545.029,Z 375.994,A -85,B 0,C 180,E1 -3698.714,E2 -3698.714} C_VEL
LIN {X 0,Y 545.165,Z 367.543,A -85,B 0,C 180,E1 -3699.647,E2 -3699.647} C_VEL
LIN {X 0,Y 545.422,Z 357.095,A -85,B 0,C 180,E1 -3700.58,E2 -3700.58} C_VEL
LIN {X 0,Y 545.606,Z 345.662,A -85,B 0,C 180,E1 -3701.4,E2 -3701.4} C_VEL
LIN {X 0,Y 545.763,Z 335.41,A -85,B 0,C 180,E1 -3701.984,E2 -3701.984} C_VEL
LIN {X 0,Y 545.977,Z 323.774,A -85,B 0,C 180,E1 -3702.498,E2 -3702.498} C_VEL
LIN {X 0,Y 546.168,Z 310.358,A -85,B 0,C 180,E1 -3702.919,E2 -3702.919} C_VEL
LIN {X 0,Y 544.759,Z 300.466,A -85,B 0,C 180,E1 -3703.166,E2 -3703.166} C_VEL
LIN {X 0,Y 544.829,Z 292.883,A -85,B 0,C 180,E1 -3705.717,E2 -3705.717} C_VEL
LIN {X 0,Y 544.859,Z 284.916,A -85,B 0,C 180,E1 -3708.422,E2 -3708.422} C_VEL
LIN {X 0,Y 544.964,Z 276.921,A -85,B 0,C 180,E1 -3711.167,E2 -3711.167} C_VEL
LIN {X 0,Y 545.014,Z 269.661,A -85,B 0,C 180,E1 -3713.715,E2 -3713.715} C_VEL
LIN {X 0,Y 545.066,Z 262.331,A -85,B 0,C 180,E1 -3716.412,E2 -3716.412} C_VEL
LIN {X 0,Y 545.266,Z 254.542,A -85,B 0,C 180,E1 -3719.326,E2 -3719.326} C_VEL
LIN {X 0,Y 545.401,Z 247.934,A -85,B 0,C 180,E1 -3721.891,E2 -3721.891} C_VEL
LIN {X 0,Y 545.51,Z 241.448,A -85,B 0,C 180,E1 -3724.531,E2 -3724.531} C_VEL
LIN {X 0,Y 545.379,Z 237.188,A -85,B 0,C 180,E1 -3726.353,E2 -3726.353} C_VEL
LIN {X 0,Y 545.109,Z 235.587,A -85,B 0,C 180,E1 -3727.134,E2 -3727.134} C_VEL
LIN {X 0,Y 545.065,Z 235.593,A -85,B 0,C 180,E1 -3730.142,E2 -3730.142} C_VEL
LIN {X 0,Y 545.085,Z 235.589,A -85,B 0,C 180,E1 -3733.105,E2 -3733.105} C_VEL
LIN {X 0,Y 545.065,Z 235.593,A -85,B 0,C 180,E1 -3736.223,E2 -3736.223} C_VEL
LIN {X 0,Y 545.099,Z 235.588,A -85,B 0,C 180,E1 -3738.886,E2 -3738.886} C_VEL
LIN {X 0,Y 545.051,Z 235.594,A -85,B 0,C 180,E1 -3741.762,E2 -3741.762} C_VEL
LIN {X 0,Y 545.062,Z 235.593,A -85,B 0,C 180,E1 -3744.533,E2 -3744.533} C_VEL
LIN {X 0,Y 545.078,Z 235.59,A -85,B 0,C 180,E1 -3747.211,E2 -3747.211} C_VEL
LIN {X 0,Y 545.098,Z 235.589,A -85,B 0,C 180,E1 -3749.812,E2 -3749.812} C_VEL
LIN {X 0,Y 545.092,Z 235.589,A -85,B 0,C 180,E1 -3752.825,E2 -3752.825} C_VEL
LIN {X 0,Y 545.047,Z 235.594,A -85,B 0,C 180,E1 -3755.63,E2 -3755.63} C_VEL
LIN {X 0,Y 545.06,Z 235.593,A -85,B 0,C 180,E1 -3758.836,E2 -3758.836} C_VEL
LIN {X 0,Y 545.079,Z 235.591,A -85,B 0,C 180,E1 -3761.195,E2 -3761.195} C_VEL
LIN {X 0,Y 545.07,Z 235.591,A -85,B 0,C 180,E1 -3763.52,E2 -3763.52} C_VEL
LIN {X 0,Y 545.09,Z 235.588,A -85,B 0,C 180,E1 -3765.819,E2 -3765.819} C_VEL
LIN {X 0,Y 545.126,Z 235.584,A -85,B 0,C 180,E1 -3768.849,E2 -3768.849} C_VEL
LIN {X 0,Y 545.128,Z 235.583,A -85,B 0,C 180,E1 -3771.846,E2 -3771.846} C_VEL
LIN {X 0,Y 545.202,Z 235.574,A -85,B 0,C 180,E1 -3774.822,E2 -3774.822} C_VEL
LIN {X 0,Y 545.187,Z 235.577,A -85,B 0,C 180,E1 -3777.783,E2 -3777.783} C_VEL
LIN {X 0,Y 545.208,Z 235.575,A -85,B 0,C 180,E1 -3780.738,E2 -3780.738} C_VEL
LIN {X 0,Y 545.169,Z 235.579,A -85,B 0,C 180,E1 -3782.955,E2 -3782.955} C_VEL
LIN {X 0,Y 545.165,Z 235.58,A -85,B 0,C 180,E1 -3785.919,E2 -3785.919} C_VEL
LIN {X 0,Y 545.119,Z 235.587,A -85,B 0,C 180,E1 -3788.899,E2 -3788.899} C_VEL
LIN {X 0,Y 545.047,Z 235.596,A -85,B 0,C 180,E1 -3790.399,E2 -3790.399} C_VEL
LIN {X 0,Y 545.062,Z 236.824,A -85,B 0,C 180,E1 -3791.502,E2 -3791.502} C_VEL
LIN {X 0,Y 544.978,Z 241.941,A -85,B 0,C 180,E1 -3794.721,E2 -3794.721} C_VEL
LIN {X 0,Y 544.897,Z 247.317,A -85,B 0,C 180,E1 -3798.031,E2 -3798.031} C_VEL
LIN {X 0,Y 544.835,Z 251.204,A -85,B 0,C 180,E1 -3800.381,E2 -3800.381} C_VEL
LIN {X 0,Y 544.824,Z 255.273,A -85,B 0,C 180,E1 -3802.766,E2 -3802.766} C_VEL
LIN {X 0,Y 544.754,Z 259.751,A -85,B 0,C 180,E1 -3805.436,E2 -3805.436} C_VEL
LIN {X 0,Y 544.705,Z 263.537,A -85,B 0,C 180,E1 -3807.676,E2 -3807.676} C_VEL
LIN {X 0,Y 544.619,Z 267.917,A -85,B 0,C 180,E1 -3810.215,E2 -3810.215} C_VEL
LIN {X 0,Y 544.619,Z 272.633,A -85,B 0,C 180,E1 -3812.903,E2 -3812.903} C_VEL
LIN {X 0,Y 546.104,Z 282.179,A -85,B 0,C 180,E1 -3813.171,E2 -3813.171} C_VEL
LIN {X 0,Y 545.931,Z 294.102,A -85,B 0,C 180,E1 -3813.557,E2 -3813.557} C_VEL
LIN {X 0,Y 545.86,Z 298.89,A -85,B 0,C 180,E1 -3813.754,E2 -3813.754} C_VEL
LIN {X 0,Y 545.121,Z 304.335,A -85,B 0,C 180,E1 -3813.985,E2 -3813.985} C_VEL
LIN {X 0,Y 542.163,Z 312.997,A -85,B 0,C 180,E1 -3814.39,E2 -3814.39} C_VEL
LIN {X 0,Y 539.186,Z 321.255,A -85,B 0,C 180,E1 -3814.876,E2 -3814.876} C_VEL
LIN {X 0,Y 538.421,Z 326.061,A -85,B 0,C 180,E1 -3815.231,E2 -3815.231} C_VEL
LIN {X 0,Y 538.138,Z 337.17,A -85,B 0,C 180,E1 -3816.224,E2 -3816.224} C_VEL
LIN {X 0,Y 537.997,Z 345.706,A -85,B 0,C 180,E1 -3817.17,E2 -3817.17} C_VEL
LIN {X 0,Y 537.761,Z 354.362,A -85,B 0,C 180,E1 -3818.36,E2 -3818.36} C_VEL
LIN {X 0,Y 537.687,Z 361.221,A -85,B 0,C 180,E1 -3819.542,E2 -3819.542} C_VEL
LIN {X 0,Y 537.597,Z 367.028,A -85,B 0,C 180,E1 -3820.816,E2 -3820.816} C_VEL
LIN {X 0,Y 537.583,Z 370.604,A -85,B 0,C 180,E1 -3821.827,E2 -3821.827} C_VEL
LIN {X 0,Y 537.486,Z 373.533,A -85,B 0,C 180,E1 -3822.927,E2 -3822.927} C_VEL
LIN {X 0,Y 537.486,Z 375.524,A -85,B 0,C 180,E1 -3824.016,E2 -3824.016} C_VEL
LIN {X 0,Y 537.494,Z 376.651,A -85,B 0,C 180,E1 -3825.085,E2 -3825.085} C_VEL
LIN {X 0,Y 537.466,Z 376.988,A -85,B 0,C 180,E1 -3826.13,E2 -3826.13} C_VEL
LIN {X 0,Y 537.455,Z 376.551,A -85,B 0,C 180,E1 -3827.159,E2 -3827.159} C_VEL
LIN {X 0,Y 537.486,Z 375.356,A -85,B 0,C 180,E1 -3828.184,E2 -3828.184} C_VEL
LIN {X 0,Y 537.482,Z 373.153,A -85,B 0,C 180,E1 -3829.321,E2 -3829.321} C_VEL
LIN {X 0,Y 537.566,Z 369.91,A -85,B 0,C 180,E1 -3830.473,E2 -3830.473} C_VEL
LIN {X 0,Y 537.601,Z 365.414,A -85,B 0,C 180,E1 -3831.661,E2 -3831.661} C_VEL
LIN {X 0,Y 537.682,Z 359.492,A -85,B 0,C 180,E1 -3832.873,E2 -3832.873} C_VEL
LIN {X 0,Y 537.807,Z 352.711,A -85,B 0,C 180,E1 -3833.982,E2 -3833.982} C_VEL
LIN {X 0,Y 537.985,Z 344.641,A -85,B 0,C 180,E1 -3835.045,E2 -3835.045} C_VEL
LIN {X 0,Y 538.199,Z 335.138,A -85,B 0,C 180,E1 -3836.063,E2 -3836.063} C_VEL
LIN {X 0,Y 538.407,Z 324.577,A -85,B 0,C 180,E1 -3836.978,E2 -3836.978} C_VEL
LIN {X 0,Y 538.605,Z 313.171,A -85,B 0,C 180,E1 -3837.759,E2 -3837.759} C_VEL
LIN {X 0,Y 538.841,Z 301.819,A -85,B 0,C 180,E1 -3838.369,E2 -3838.369} C_VEL
LIN {X 0,Y 539.063,Z 290.271,A -85,B 0,C 180,E1 -3838.841,E2 -3838.841} C_VEL
LIN {X 0,Y 539.03,Z 281.529,A -85,B 0,C 180,E1 -3839.112,E2 -3839.112} C_VEL
LIN {X 0,Y 537.525,Z 272.773,A -85,B 0,C 180,E1 -3839.366,E2 -3839.366} C_VEL
LIN {X 0,Y 537.557,Z 266.822,A -85,B 0,C 180,E1 -3842.769,E2 -3842.769} C_VEL
LIN {X 0,Y 537.596,Z 262.543,A -85,B 0,C 180,E1 -3845.271,E2 -3845.271} C_VEL
LIN {X 0,Y 537.699,Z 256.998,A -85,B 0,C 180,E1 -3848.533,E2 -3848.533} C_VEL
LIN {X 0,Y 537.744,Z 252.957,A -85,B 0,C 180,E1 -3850.93,E2 -3850.93} C_VEL
LIN {X 0,Y 537.783,Z 249.07,A -85,B 0,C 180,E1 -3853.292,E2 -3853.292} C_VEL
LIN {X 0,Y 537.852,Z 245.275,A -85,B 0,C 180,E1 -3855.625,E2 -3855.625} C_VEL
LIN {X 0,Y 537.982,Z 240.324,A -85,B 0,C 180,E1 -3858.7,E2 -3858.7} C_VEL
LIN {X 0,Y 537.95,Z 236.732,A -85,B 0,C 180,E1 -3860.981,E2 -3860.981} C_VEL
LIN {X 0,Y 538.12,Z 236.456,A -85,B 0,C 180,E1 -3863.005,E2 -3863.005} C_VEL
LIN {X 0,Y 538.153,Z 236.454,A -85,B 0,C 180,E1 -3864.755,E2 -3864.755} C_VEL
LIN {X 0,Y 538.155,Z 236.45,A -85,B 0,C 180,E1 -3867.755,E2 -3867.755} C_VEL
LIN {X 0,Y 538.176,Z 236.451,A -85,B 0,C 180,E1 -3870.748,E2 -3870.748} C_VEL
LIN {X 0,Y 538.133,Z 236.456,A -85,B 0,C 180,E1 -3872.995,E2 -3872.995} C_VEL
LIN {X 0,Y 538.114,Z 236.457,A -85,B 0,C 180,E1 -3875.997,E2 -3875.997} C_VEL
LIN {X 0,Y 538.069,Z 236.464,A -85,B 0,C 180,E1 -3879.018,E2 -3879.018} C_VEL
LIN {X 0,Y 538.073,Z 236.462,A -85,B 0,C 180,E1 -3882.063,E2 -3882.063} C_VEL
LIN {X 0,Y 538.035,Z 236.468,A -85,B 0,C 180,E1 -3885.144,E2 -3885.144} C_VEL
LIN {X 0,Y 538.025,Z 236.468,A -85,B 0,C 180,E1 -3888.27,E2 -3888.27} C_VEL
LIN {X 0,Y 538.032,Z 236.466,A -85,B 0,C 180,E1 -3890.651,E2 -3890.651} C_VEL
LIN {X 0,Y 538.03,Z 236.468,A -85,B 0,C 180,E1 -3893.887,E2 -3893.887} C_VEL
LIN {X 0,Y 538.039,Z 236.466,A -85,B 0,C 180,E1 -3896.366,E2 -3896.366} C_VEL
LIN {X 0,Y 538.045,Z 236.464,A -85,B 0,C 180,E1 -3898.939,E2 -3898.939} C_VEL
LIN {X 0,Y 538.017,Z 236.471,A -85,B 0,C 180,E1 -3901.891,E2 -3901.891} C_VEL
LIN {X 0,Y 538.02,Z 236.469,A -85,B 0,C 180,E1 -3904.621,E2 -3904.621} C_VEL
LIN {X 0,Y 537.997,Z 236.472,A -85,B 0,C 180,E1 -3907.171,E2 -3907.171} C_VEL
LIN {X 0,Y 538.044,Z 236.465,A -85,B 0,C 180,E1 -3909.794,E2 -3909.794} C_VEL
LIN {X 0,Y 538.014,Z 236.47,A -85,B 0,C 180,E1 -3912.786,E2 -3912.786} C_VEL
LIN {X 0,Y 538.018,Z 236.468,A -85,B 0,C 180,E1 -3915.926,E2 -3915.926} C_VEL
LIN {X 0,Y 538.067,Z 236.463,A -85,B 0,C 180,E1 -3919.249,E2 -3919.249} C_VEL
LIN {X 0,Y 537.984,Z 236.473,A -85,B 0,C 180,E1 -3922.123,E2 -3922.123} C_VEL
LIN {X 0,Y 538.009,Z 236.472,A -85,B 0,C 180,E1 -3924.918,E2 -3924.918} C_VEL
LIN {X 0,Y 538.021,Z 236.468,A -85,B 0,C 180,E1 -3927.619,E2 -3927.619} C_VEL
LIN {X 0,Y 538.032,Z 236.466,A -85,B 0,C 180,E1 -3930.241,E2 -3930.241} C_VEL
LIN {X 0,Y 538.061,Z 236.463,A -85,B 0,C 180,E1 -3932.797,E2 -3932.797} C_VEL
LIN {X 0,Y 538.04,Z 236.466,A -85,B 0,C 180,E1 -3935.293,E2 -3935.293} C_VEL
LIN {X 0,Y 538.005,Z 236.472,A -85,B 0,C 180,E1 -3938.042,E2 -3938.042} C_VEL
LIN {X 0,Y 538.031,Z 236.467,A -85,B 0,C 180,E1 -3940.941,E2 -3940.941} C_VEL
LIN {X 0,Y 538.018,Z 236.468,A -85,B 0,C 180,E1 -3943.3,E2 -3943.3} C_VEL
LIN {X 0,Y 538.055,Z 236.463,A -85,B 0,C 180,E1 -3945.631,E2 -3945.631} C_VEL
LIN {X 0,Y 538.082,Z 236.463,A -85,B 0,C 180,E1 -3948.703,E2 -3948.703} C_VEL
LIN {X 0,Y 538.083,Z 236.46,A -85,B 0,C 180,E1 -3951.741,E2 -3951.741} C_VEL
LIN {X 0,Y 538.156,Z 236.454,A -85,B 0,C 180,E1 -3954.756,E2 -3954.756} C_VEL
LIN {X 0,Y 538.161,Z 236.45,A -85,B 0,C 180,E1 -3957.756,E2 -3957.756} C_VEL
LIN {X 0,Y 538.179,Z 236.451,A -85,B 0,C 180,E1 -3960.749,E2 -3960.749} C_VEL
LIN {X 0,Y 538.133,Z 236.455,A -85,B 0,C 180,E1 -3962.995,E2 -3962.995} C_VEL
LIN {X 0,Y 538.117,Z 236.457,A -85,B 0,C 180,E1 -3965.998,E2 -3965.998} C_VEL
LIN {X 0,Y 538.063,Z 236.464,A -85,B 0,C 180,E1 -3969.019,E2 -3969.019} C_VEL
LIN {X 0,Y 538.078,Z 236.461,A -85,B 0,C 180,E1 -3972.063,E2 -3972.063} C_VEL
LIN {X 0,Y 538.04,Z 236.467,A -85,B 0,C 180,E1 -3975.145,E2 -3975.145} C_VEL
LIN {X 0,Y 538.027,Z 236.467,A -85,B 0,C 180,E1 -3978.271,E2 -3978.271} C_VEL
LIN {X 0,Y 538.035,Z 236.465,A -85,B 0,C 180,E1 -3980.652,E2 -3980.652} C_VEL
LIN {X 0,Y 538.021,Z 236.469,A -85,B 0,C 180,E1 -3983.888,E2 -3983.888} C_VEL
LIN {X 0,Y 538.039,Z 236.465,A -85,B 0,C 180,E1 -3986.368,E2 -3986.368} C_VEL
LIN {X 0,Y 538.028,Z 236.467,A -85,B 0,C 180,E1 -3988.935,E2 -3988.935} C_VEL
LIN {X 0,Y 538.007,Z 236.472,A -85,B 0,C 180,E1 -3991.888,E2 -3991.888} C_VEL
LIN {X 0,Y 538.024,Z 236.469,A -85,B 0,C 180,E1 -3994.621,E2 -3994.621} C_VEL
LIN {X 0,Y 538.004,Z 236.471,A -85,B 0,C 180,E1 -3997.171,E2 -3997.171} C_VEL
LIN {X 0,Y 538.025,Z 236.467,A -85,B 0,C 180,E1 -3999.797,E2 -3999.797} C_VEL
LIN {X 0,Y 538.018,Z 236.47,A -85,B 0,C 180,E1 -4002.787,E2 -4002.787} C_VEL
LIN {X 0,Y 538.018,Z 236.468,A -85,B 0,C 180,E1 -4005.927,E2 -4005.927} C_VEL
LIN {X 0,Y 538.052,Z 236.464,A -85,B 0,C 180,E1 -4009.225,E2 -4009.225} C_VEL
LIN {X 0,Y 538.039,Z 236.468,A -85,B 0,C 180,E1 -4012.51,E2 -4012.51} C_VEL
LIN {X 0,Y 538.063,Z 236.525,A -85,B 0,C 180,E1 -4012.823,E2 -4012.823} C_VEL
LIN {X 0,Y 538.572,Z 240.391,A -85,B 0,C 180,E1 -4014.501,E2 -4014.501} C_VEL
LIN {X 0,Y 538.456,Z 246.967,A -85,B 0,C 180,E1 -4017.204,E2 -4017.204} C_VEL
LIN {X 0,Y 538.284,Z 254.682,A -85,B 0,C 180,E1 -4020.256,E2 -4020.256} C_VEL
LIN {X 0,Y 538.077,Z 262.401,A -85,B 0,C 180,E1 -4023.217,E2 -4023.217} C_VEL
LIN {X 0,Y 538.01,Z 270.239,A -85,B 0,C 180,E1 -4026.123,E2 -4026.123} C_VEL
LIN {X 0,Y 537.913,Z 278.148,A -85,B 0,C 180,E1 -4028.943,E2 -4028.943} C_VEL
LIN {X 0,Y 537.829,Z 286.066,A -85,B 0,C 180,E1 -4031.723,E2 -4031.723} C_VEL
LIN {X 0,Y 537.775,Z 293.964,A -85,B 0,C 180,E1 -4034.46,E2 -4034.46} C_VEL
LIN {X 0,Y 537.694,Z 300.575,A -85,B 0,C 180,E1 -4036.669,E2 -4036.669} C_VEL
LIN {X 0,Y 539.221,Z 311.051,A -85,B 0,C 180,E1 -4036.935,E2 -4036.935} C_VEL
LIN {X 0,Y 539.029,Z 323.58,A -85,B 0,C 180,E1 -4037.338,E2 -4037.338} C_VEL
LIN {X 0,Y 538.815,Z 335.247,A -85,B 0,C 180,E1 -4037.859,E2 -4037.859} C_VEL
LIN {X 0,Y 538.553,Z 347.67,A -85,B 0,C 180,E1 -4038.591,E2 -4038.591} C_VEL
LIN {X 0,Y 538.406,Z 358.188,A -85,B 0,C 180,E1 -4039.375,E2 -4039.375} C_VEL
LIN {X 0,Y 538.137,Z 367.501,A -85,B 0,C 180,E1 -4040.225,E2 -4040.225} C_VEL
LIN {X 0,Y 537.974,Z 375.99,A -85,B 0,C 180,E1 -4041.17,E2 -4041.17} C_VEL
LIN {X 0,Y 537.817,Z 384.235,A -85,B 0,C 180,E1 -4042.303,E2 -4042.303} C_VEL
LIN {X 0,Y 537.684,Z 390.751,A -85,B 0,C 180,E1 -4043.409,E2 -4043.409} C_VEL
LIN {X 0,Y 537.677,Z 395.366,A -85,B 0,C 180,E1 -4044.374,E2 -4044.374} C_VEL
LIN {X 0,Y 537.558,Z 399.676,A -85,B 0,C 180,E1 -4045.501,E2 -4045.501} C_VEL
LIN {X 0,Y 537.591,Z 401.958,A -85,B 0,C 180,E1 -4046.252,E2 -4046.252} C_VEL
LIN {X 0,Y 537.551,Z 403.806,A -85,B 0,C 180,E1 -4047.002,E2 -4047.002} C_VEL
LIN {X 0,Y 537.451,Z 406.182,A -85,B 0,C 180,E1 -4048.501,E2 -4048.501} C_VEL
LIN {X 0,Y 537.442,Z 407,A -85,B 0,C 180,E1 -4050,E2 -4050} C_VEL
LIN {X 0,Y 537.452,Z 406.183,A -85,B 0,C 180,E1 -4051.498,E2 -4051.498} C_VEL
LIN {X 0,Y 537.551,Z 403.81,A -85,B 0,C 180,E1 -4052.998,E2 -4052.998} C_VEL
LIN {X 0,Y 537.604,Z 400.896,A -85,B 0,C 180,E1 -4054.123,E2 -4054.123} C_VEL
LIN {X 0,Y 537.588,Z 396.949,A -85,B 0,C 180,E1 -4055.25,E2 -4055.25} C_VEL
LIN {X 0,Y 537.645,Z 392.128,A -85,B 0,C 180,E1 -4056.326,E2 -4056.326} C_VEL
LIN {X 0,Y 537.791,Z 385.468,A -85,B 0,C 180,E1 -4057.509,E2 -4057.509} C_VEL
LIN {X 0,Y 537.973,Z 377.479,A -85,B 0,C 180,E1 -4058.64,E2 -4058.64} C_VEL
LIN {X 0,Y 538.119,Z 369.302,A -85,B 0,C 180,E1 -4059.585,E2 -4059.585} C_VEL
LIN {X 0,Y 538.377,Z 359.32,A -85,B 0,C 180,E1 -4060.53,E2 -4060.53} C_VEL
LIN {X 0,Y 538.521,Z 349.47,A -85,B 0,C 180,E1 -4061.289,E2 -4061.289} C_VEL
LIN {X 0,Y 538.715,Z 338.43,A -85,B 0,C 180,E1 -4061.971,E2 -4061.971} C_VEL
LIN {X 0,Y 538.962,Z 325.891,A -85,B 0,C 180,E1 -4062.568,E2 -4062.568} C_VEL
LIN {X 0,Y 539.18,Z 312.841,A -85,B 0,C 180,E1 -4063.017,E2 -4063.017} C_VEL
LIN {X 0,Y 538.905,Z 307.769,A -85,B 0,C 180,E1 -4063.156,E2 -4063.156} C_VEL
LIN {X 0,Y 537.671,Z 300.296,A -85,B 0,C 180,E1 -4063.343,E2 -4063.343} C_VEL
LIN {X 0,Y 537.773,Z 291.575,A -85,B 0,C 180,E1 -4066.318,E2 -4066.318} C_VEL
LIN {X 0,Y 537.832,Z 283.602,A -85,B 0,C 180,E1 -4069.067,E2 -4069.067} C_VEL
LIN {X 0,Y 537.919,Z 275.398,A -85,B 0,C 180,E1 -4071.931,E2 -4071.931} C_VEL
LIN {X 0,Y 538.022,Z 266.674,A -85,B 0,C 180,E1 -4075.121,E2 -4075.121} C_VEL
LIN {X 0,Y 538.151,Z 257.77,A -85,B 0,C 180,E1 -4078.468,E2 -4078.468} C_VEL
LIN {X 0,Y 538.355,Z 250.065,A -85,B 0,C 180,E1 -4081.478,E2 -4081.478} C_VEL
LIN {X 0,Y 538.498,Z 243.587,A -85,B 0,C 180,E1 -4084.138,E2 -4084.138} C_VEL
LIN {X 0,Y 538.514,Z 239.262,A -85,B 0,C 180,E1 -4085.987,E2 -4085.987} C_VEL
LIN {X 0,Y 538.057,Z 236.464,A -85,B 0,C 180,E1 -4087.304,E2 -4087.304} C_VEL
LIN {X 0,Y 538.048,Z 236.466,A -85,B 0,C 180,E1 -4090.746,E2 -4090.746} C_VEL
LIN {X 0,Y 538.017,Z 236.469,A -85,B 0,C 180,E1 -4093.813,E2 -4093.813} C_VEL
LIN {X 0,Y 538.018,Z 236.47,A -85,B 0,C 180,E1 -4096.185,E2 -4096.185} C_VEL
LIN {X 0,Y 538.076,Z 236.463,A -85,B 0,C 180,E1 -4099.248,E2 -4099.248} C_VEL
LIN {X 0,Y 537.999,Z 236.472,A -85,B 0,C 180,E1 -4102.122,E2 -4102.122} C_VEL
LIN {X 0,Y 538.017,Z 236.47,A -85,B 0,C 180,E1 -4104.916,E2 -4104.916} C_VEL
LIN {X 0,Y 538.028,Z 236.469,A -85,B 0,C 180,E1 -4107.617,E2 -4107.617} C_VEL
LIN {X 0,Y 538.039,Z 236.466,A -85,B 0,C 180,E1 -4110.239,E2 -4110.239} C_VEL
LIN {X 0,Y 538.062,Z 236.465,A -85,B 0,C 180,E1 -4112.795,E2 -4112.795} C_VEL
LIN {X 0,Y 538.044,Z 236.466,A -85,B 0,C 180,E1 -4115.292,E2 -4115.292} C_VEL
LIN {X 0,Y 538.009,Z 236.472,A -85,B 0,C 180,E1 -4118.041,E2 -4118.041} C_VEL
LIN {X 0,Y 538.035,Z 236.468,A -85,B 0,C 180,E1 -4120.939,E2 -4120.939} C_VEL
LIN {X 0,Y 538.021,Z 236.47,A -85,B 0,C 180,E1 -4123.298,E2 -4123.298} C_VEL
LIN {X 0,Y 538.058,Z 236.464,A -85,B 0,C 180,E1 -4125.63,E2 -4125.63} C_VEL
LIN {X 0,Y 538.083,Z 236.461,A -85,B 0,C 180,E1 -4128.701,E2 -4128.701} C_VEL
LIN {X 0,Y 538.085,Z 236.461,A -85,B 0,C 180,E1 -4131.739,E2 -4131.739} C_VEL
LIN {X 0,Y 538.159,Z 236.451,A -85,B 0,C 180,E1 -4134.754,E2 -4134.754} C_VEL
LIN {X 0,Y 538.159,Z 236.452,A -85,B 0,C 180,E1 -4137.754,E2 -4137.754} C_VEL
LIN {X 0,Y 538.177,Z 236.45,A -85,B 0,C 180,E1 -4140.747,E2 -4140.747} C_VEL
LIN {X 0,Y 538.135,Z 236.456,A -85,B 0,C 180,E1 -4142.994,E2 -4142.994} C_VEL
LIN {X 0,Y 538.118,Z 236.458,A -85,B 0,C 180,E1 -4145.996,E2 -4145.996} C_VEL
LIN {X 0,Y 538.067,Z 236.464,A -85,B 0,C 180,E1 -4149.017,E2 -4149.017} C_VEL
LIN {X 0,Y 537.985,Z 236.476,A -85,B 0,C 180,E1 -4150.537,E2 -4150.537} C_VEL
LIN {X 0,Y 537.968,Z 238.6,A -85,B 0,C 180,E1 -4152.064,E2 -4152.064} C_VEL
LIN {X 0,Y 537.936,Z 243.458,A -85,B 0,C 180,E1 -4155.146,E2 -4155.146} C_VEL
LIN {X 0,Y 537.822,Z 248.496,A -85,B 0,C 180,E1 -4158.276,E2 -4158.276} C_VEL
LIN {X 0,Y 537.783,Z 252.383,A -85,B 0,C 180,E1 -4160.66,E2 -4160.66} C_VEL
LIN {X 0,Y 537.724,Z 256.442,A -85,B 0,C 180,E1 -4163.084,E2 -4163.084} C_VEL
LIN {X 0,Y 537.678,Z 260.658,A -85,B 0,C 180,E1 -4165.594,E2 -4165.594} C_VEL
LIN {X 0,Y 537.624,Z 264.803,A -85,B 0,C 180,E1 -4168.072,E2 -4168.072} C_VEL
LIN {X 0,Y 537.55,Z 270.722,A -85,B 0,C 180,E1 -4171.53,E2 -4171.53} C_VEL
LIN {X 0,Y 537.52,Z 272.798,A -85,B 0,C 180,E1 -4172.721,E2 -4172.721} C_VEL
LIN {X 0,Y 539.163,Z 283.198,A -85,B 0,C 180,E1 -4173.025,E2 -4173.025} C_VEL
LIN {X 0,Y 538.999,Z 295.362,A -85,B 0,C 180,E1 -4173.439,E2 -4173.439} C_VEL
LIN {X 0,Y 538.758,Z 307.686,A -85,B 0,C 180,E1 -4174.017,E2 -4174.017} C_VEL
LIN {X 0,Y 538.56,Z 318.948,A -85,B 0,C 180,E1 -4174.704,E2 -4174.704} C_VEL
LIN {X 0,Y 538.421,Z 326.061,A -85,B 0,C 180,E1 -4175.231,E2 -4175.231} C_VEL
LIN {X 0,Y 537.662,Z 330.792,A -85,B 0,C 180,E1 -4175.611,E2 -4175.611} C_VEL
LIN {X 0,Y 534.678,Z 338.146,A -85,B 0,C 180,E1 -4176.25,E2 -4176.25} C_VEL
LIN {X 0,Y 531.676,Z 344.932,A -85,B 0,C 180,E1 -4176.951,E2 -4176.951} C_VEL
LIN {X 0,Y 530.889,Z 348.765,A -85,B 0,C 180,E1 -4177.423,E2 -4177.423} C_VEL
LIN {X 0,Y 530.714,Z 356.034,A -85,B 0,C 180,E1 -4178.49,E2 -4178.49} C_VEL
LIN {X 0,Y 530.614,Z 361.52,A -85,B 0,C 180,E1 -4179.475,E2 -4179.475} C_VEL
LIN {X 0,Y 530.522,Z 366.092,A -85,B 0,C 180,E1 -4180.474,E2 -4180.474} C_VEL
LIN {X 0,Y 530.494,Z 369.818,A -85,B 0,C 180,E1 -4181.482,E2 -4181.482} C_VEL
LIN {X 0,Y 530.429,Z 372.789,A -85,B 0,C 180,E1 -4182.509,E2 -4182.509} C_VEL
LIN {X 0,Y 530.363,Z 374.989,A -85,B 0,C 180,E1 -4183.555,E2 -4183.555} C_VEL
LIN {X 0,Y 530.391,Z 376.387,A -85,B 0,C 180,E1 -4184.608,E2 -4184.608} C_VEL
LIN {X 0,Y 530.389,Z 377.044,A -85,B 0,C 180,E1 -4185.685,E2 -4185.685} C_VEL
LIN {X 0,Y 530.333,Z 376.91,A -85,B 0,C 180,E1 -4186.789,E2 -4186.789} C_VEL
LIN {X 0,Y 530.381,Z 375.929,A -85,B 0,C 180,E1 -4187.904,E2 -4187.904} C_VEL
LIN {X 0,Y 530.39,Z 374.007,A -85,B 0,C 180,E1 -4189.048,E2 -4189.048} C_VEL
LIN {X 0,Y 530.481,Z 370.122,A -85,B 0,C 180,E1 -4190.513,E2 -4190.513} C_VEL
LIN {X 0,Y 530.543,Z 365.576,A -85,B 0,C 180,E1 -4191.737,E2 -4191.737} C_VEL
LIN {X 0,Y 530.631,Z 359.348,A -85,B 0,C 180,E1 -4193.026,E2 -4193.026} C_VEL
LIN {X 0,Y 530.764,Z 352.646,A -85,B 0,C 180,E1 -4194.123,E2 -4194.123} C_VEL
LIN {X 0,Y 531.004,Z 343.564,A -85,B 0,C 180,E1 -4195.312,E2 -4195.312} C_VEL
LIN {X 0,Y 531.207,Z 334.815,A -85,B 0,C 180,E1 -4196.244,E2 -4196.244} C_VEL
LIN {X 0,Y 531.453,Z 324.135,A -85,B 0,C 180,E1 -4197.168,E2 -4197.168} C_VEL
LIN {X 0,Y 531.66,Z 312.378,A -85,B 0,C 180,E1 -4197.972,E2 -4197.972} C_VEL
LIN {X 0,Y 531.926,Z 300.622,A -85,B 0,C 180,E1 -4198.597,E2 -4198.597} C_VEL
LIN {X 0,Y 532.212,Z 287.528,A -85,B 0,C 180,E1 -4199.106,E2 -4199.106} C_VEL
LIN {X 0,Y 532.04,Z 281.902,A -85,B 0,C 180,E1 -4199.28,E2 -4199.28} C_VEL
LIN {X 0,Y 530.443,Z 272.965,A -85,B 0,C 180,E1 -4199.546,E2 -4199.546} C_VEL
LIN {X 0,Y 530.474,Z 267.735,A -85,B 0,C 180,E1 -4202.576,E2 -4202.576} C_VEL
LIN {X 0,Y 530.511,Z 263.74,A -85,B 0,C 180,E1 -4204.918,E2 -4204.918} C_VEL
LIN {X 0,Y 530.573,Z 259.509,A -85,B 0,C 180,E1 -4207.41,E2 -4207.41} C_VEL
LIN {X 0,Y 530.688,Z 255.039,A -85,B 0,C 180,E1 -4210.092,E2 -4210.092} C_VEL
LIN {X 0,Y 530.709,Z 250.17,A -85,B 0,C 180,E1 -4213.062,E2 -4213.062} C_VEL
LIN {X 0,Y 530.789,Z 246.346,A -85,B 0,C 180,E1 -4215.43,E2 -4215.43} C_VEL
LIN {X 0,Y 530.939,Z 241.372,A -85,B 0,C 180,E1 -4218.548,E2 -4218.548} C_VEL
LIN {X 0,Y 530.9,Z 237.767,A -85,B 0,C 180,E1 -4220.86,E2 -4220.86} C_VEL
LIN {X 0,Y 530.958,Z 237.345,A -85,B 0,C 180,E1 -4221.628,E2 -4221.628} C_VEL
LIN {X 0,Y 531.074,Z 237.334,A -85,B 0,C 180,E1 -4223.923,E2 -4223.923} C_VEL
LIN {X 0,Y 531.098,Z 237.332,A -85,B 0,C 180,E1 -4226.966,E2 -4226.966} C_VEL
LIN {X 0,Y 531.131,Z 237.327,A -85,B 0,C 180,E1 -4230,E2 -4230} C_VEL
LIN {X 0,Y 531.099,Z 237.332,A -85,B 0,C 180,E1 -4233.034,E2 -4233.034} C_VEL
LIN {X 0,Y 531.074,Z 237.334,A -85,B 0,C 180,E1 -4236.077,E2 -4236.077} C_VEL
LIN {X 0,Y 531.028,Z 237.341,A -85,B 0,C 180,E1 -4239.138,E2 -4239.138} C_VEL
LIN {X 0,Y 531.03,Z 237.339,A -85,B 0,C 180,E1 -4242.225,E2 -4242.225} C_VEL
LIN {X 0,Y 530.986,Z 237.346,A -85,B 0,C 180,E1 -4245.35,E2 -4245.35} C_VEL
LIN {X 0,Y 531.006,Z 237.344,A -85,B 0,C 180,E1 -4247.722,E2 -4247.722} C_VEL
LIN {X 0,Y 530.994,Z 237.344,A -85,B 0,C 180,E1 -4250.938,E2 -4250.938} C_VEL
LIN {X 0,Y 530.997,Z 237.343,A -85,B 0,C 180,E1 -4254.045,E2 -4254.045} C_VEL
LIN {X 0,Y 531.001,Z 237.342,A -85,B 0,C 180,E1 -4256.743,E2 -4256.743} C_VEL
LIN {X 0,Y 530.989,Z 237.344,A -85,B 0,C 180,E1 -4259.322,E2 -4259.322} C_VEL
LIN {X 0,Y 530.97,Z 237.348,A -85,B 0,C 180,E1 -4262.103,E2 -4262.103} C_VEL
LIN {X 0,Y 530.977,Z 237.345,A -85,B 0,C 180,E1 -4264.854,E2 -4264.854} C_VEL
LIN {X 0,Y 530.956,Z 237.348,A -85,B 0,C 180,E1 -4267.508,E2 -4267.508} C_VEL
LIN {X 0,Y 531.015,Z 237.342,A -85,B 0,C 180,E1 -4270.429,E2 -4270.429} C_VEL
LIN {X 0,Y 530.956,Z 237.348,A -85,B 0,C 180,E1 -4273.495,E2 -4273.495} C_VEL
LIN {X 0,Y 530.957,Z 237.35,A -85,B 0,C 180,E1 -4276.506,E2 -4276.506} C_VEL
LIN {X 0,Y 530.997,Z 237.343,A -85,B 0,C 180,E1 -4279.57,E2 -4279.57} C_VEL
LIN {X 0,Y 530.959,Z 237.35,A -85,B 0,C 180,E1 -4282.577,E2 -4282.577} C_VEL
LIN {X 0,Y 530.99,Z 237.344,A -85,B 0,C 180,E1 -4285.312,E2 -4285.312} C_VEL
LIN {X 0,Y 530.972,Z 237.346,A -85,B 0,C 180,E1 -4288.034,E2 -4288.034} C_VEL
LIN {X 0,Y 530.997,Z 237.346,A -85,B 0,C 180,E1 -4290.871,E2 -4290.871} C_VEL
LIN {X 0,Y 531.002,Z 237.344,A -85,B 0,C 180,E1 -4293.257,E2 -4293.257} C_VEL
LIN {X 0,Y 530.987,Z 237.344,A -85,B 0,C 180,E1 -4295.958,E2 -4295.958} C_VEL
LIN {X 0,Y 530.993,Z 237.345,A -85,B 0,C 180,E1 -4299.063,E2 -4299.063} C_VEL
LIN {X 0,Y 531.007,Z 237.341,A -85,B 0,C 180,E1 -4302.278,E2 -4302.278} C_VEL
LIN {X 0,Y 531.01,Z 237.342,A -85,B 0,C 180,E1 -4305.437,E2 -4305.437} C_VEL
LIN {X 0,Y 531.039,Z 237.339,A -85,B 0,C 180,E1 -4308.551,E2 -4308.551} C_VEL
LIN {X 0,Y 531.052,Z 237.336,A -85,B 0,C 180,E1 -4311.63,E2 -4311.63} C_VEL
LIN {X 0,Y 531.115,Z 237.33,A -85,B 0,C 180,E1 -4314.686,E2 -4314.686} C_VEL
LIN {X 0,Y 531.133,Z 237.326,A -85,B 0,C 180,E1 -4317.726,E2 -4317.726} C_VEL
LIN {X 0,Y 531.149,Z 237.326,A -85,B 0,C 180,E1 -4320.759,E2 -4320.759} C_VEL
LIN {X 0,Y 531.1,Z 237.332,A -85,B 0,C 180,E1 -4323.035,E2 -4323.035} C_VEL
LIN {X 0,Y 531.077,Z 237.333,A -85,B 0,C 180,E1 -4326.078,E2 -4326.078} C_VEL
LIN {X 0,Y 531.024,Z 237.341,A -85,B 0,C 180,E1 -4329.139,E2 -4329.139} C_VEL
LIN {X 0,Y 531.036,Z 237.338,A -85,B 0,C 180,E1 -4332.226,E2 -4332.226} C_VEL
LIN {X 0,Y 530.991,Z 237.346,A -85,B 0,C 180,E1 -4335.351,E2 -4335.351} C_VEL
LIN {X 0,Y 530.986,Z 237.345,A -85,B 0,C 180,E1 -4338.522,E2 -4338.522} C_VEL
LIN {X 0,Y 530.995,Z 237.343,A -85,B 0,C 180,E1 -4340.939,E2 -4340.939} C_VEL
LIN {X 0,Y 530.976,Z 237.345,A -85,B 0,C 180,E1 -4344.225,E2 -4344.225} C_VEL
LIN {X 0,Y 531.002,Z 237.341,A -85,B 0,C 180,E1 -4346.745,E2 -4346.745} C_VEL
LIN {X 0,Y 530.979,Z 237.346,A -85,B 0,C 180,E1 -4349.324,E2 -4349.324} C_VEL
LIN {X 0,Y 530.962,Z 237.348,A -85,B 0,C 180,E1 -4352.101,E2 -4352.101} C_VEL
LIN {X 0,Y 530.982,Z 237.345,A -85,B 0,C 180,E1 -4354.854,E2 -4354.854} C_VEL
LIN {X 0,Y 530.965,Z 237.347,A -85,B 0,C 180,E1 -4357.508,E2 -4357.508} C_VEL
LIN {X 0,Y 530.982,Z 237.346,A -85,B 0,C 180,E1 -4360.434,E2 -4360.434} C_VEL
LIN {X 0,Y 530.96,Z 237.348,A -85,B 0,C 180,E1 -4363.282,E2 -4363.282} C_VEL
LIN {X 0,Y 530.981,Z 237.345,A -85,B 0,C 180,E1 -4365.622,E2 -4365.622} C_VEL
LIN {X 0,Y 531,Z 237.343,A -85,B 0,C 180,E1 -4368.566,E2 -4368.566} C_VEL
LIN {X 0,Y 530.958,Z 237.349,A -85,B 0,C 180,E1 -4371.53,E2 -4371.53} C_VEL
LIN {X 0,Y 531.03,Z 237.379,A -85,B 0,C 180,E1 -4372.639,E2 -4372.639} C_VEL
LIN {X 0,Y 531.557,Z 241.43,A -85,B 0,C 180,E1 -4374.427,E2 -4374.427} C_VEL
LIN {X 0,Y 531.467,Z 248.013,A -85,B 0,C 180,E1 -4377.169,E2 -4377.169} C_VEL
LIN {X 0,Y 531.275,Z 255.716,A -85,B 0,C 180,E1 -4380.26,E2 -4380.26} C_VEL
LIN {X 0,Y 531.041,Z 263.468,A -85,B 0,C 180,E1 -4383.259,E2 -4383.259} C_VEL
LIN {X 0,Y 530.957,Z 270.629,A -85,B 0,C 180,E1 -4385.969,E2 -4385.969} C_VEL
LIN {X 0,Y 530.846,Z 279.171,A -85,B 0,C 180,E1 -4389.056,E2 -4389.056} C_VEL
LIN {X 0,Y 530.77,Z 287.087,A -85,B 0,C 180,E1 -4391.871,E2 -4391.871} C_VEL
LIN {X 0,Y 530.673,Z 294.973,A -85,B 0,C 180,E1 -4394.641,E2 -4394.641} C_VEL
LIN {X 0,Y 530.619,Z 300.325,A -85,B 0,C 180,E1 -4396.488,E2 -4396.488} C_VEL
LIN {X 0,Y 532.311,Z 311.726,A -85,B 0,C 180,E1 -4396.787,E2 -4396.787} C_VEL
LIN {X 0,Y 532.071,Z 324.558,A -85,B 0,C 180,E1 -4397.218,E2 -4397.218} C_VEL
LIN {X 0,Y 531.828,Z 336.785,A -85,B 0,C 180,E1 -4397.794,E2 -4397.794} C_VEL
LIN {X 0,Y 531.556,Z 347.655,A -85,B 0,C 180,E1 -4398.453,E2 -4398.453} C_VEL
LIN {X 0,Y 531.354,Z 359.104,A -85,B 0,C 180,E1 -4399.329,E2 -4399.329} C_VEL
LIN {X 0,Y 531.071,Z 369.084,A -85,B 0,C 180,E1 -4400.286,E2 -4400.286} C_VEL
LIN {X 0,Y 530.887,Z 378.763,A -85,B 0,C 180,E1 -4401.435,E2 -4401.435} C_VEL
LIN {X 0,Y 530.682,Z 386.465,A -85,B 0,C 180,E1 -4402.581,E2 -4402.581} C_VEL
LIN {X 0,Y 530.605,Z 393.566,A -85,B 0,C 180,E1 -4403.917,E2 -4403.917} C_VEL
LIN {X 0,Y 530.459,Z 398.286,A -85,B 0,C 180,E1 -4405.06,E2 -4405.06} C_VEL
LIN {X 0,Y 530.516,Z 401.896,A -85,B 0,C 180,E1 -4406.202,E2 -4406.202} C_VEL
LIN {X 0,Y 530.457,Z 403.755,A -85,B 0,C 180,E1 -4406.962,E2 -4406.962} C_VEL
LIN {X 0,Y 530.412,Z 405.149,A -85,B 0,C 180,E1 -4407.722,E2 -4407.722} C_VEL
LIN {X 0,Y 530.344,Z 406.75,A -85,B 0,C 180,E1 -4409.241,E2 -4409.241} C_VEL
LIN {X 0,Y 530.343,Z 406.967,A -85,B 0,C 180,E1 -4410,E2 -4410} C_VEL
LIN {X 0,Y 530.361,Z 406.145,A -85,B 0,C 180,E1 -4411.519,E2 -4411.519} C_VEL
LIN {X 0,Y 530.412,Z 405.152,A -85,B 0,C 180,E1 -4412.278,E2 -4412.278} C_VEL
LIN {X 0,Y 530.457,Z 403.758,A -85,B 0,C 180,E1 -4413.038,E2 -4413.038} C_VEL
LIN {X 0,Y 530.523,Z 400.824,A -85,B 0,C 180,E1 -4414.178,E2 -4414.178} C_VEL
LIN {X 0,Y 530.525,Z 396.85,A -85,B 0,C 180,E1 -4415.321,E2 -4415.321} C_VEL
LIN {X 0,Y 530.597,Z 391.144,A -85,B 0,C 180,E1 -4416.578,E2 -4416.578} C_VEL
LIN {X 0,Y 530.734,Z 384.055,A -85,B 0,C 180,E1 -4417.801,E2 -4417.801} C_VEL
LIN {X 0,Y 530.931,Z 375.762,A -85,B 0,C 180,E1 -4418.948,E2 -4418.948} C_VEL
LIN {X 0,Y 531.098,Z 367.258,A -85,B 0,C 180,E1 -4419.905,E2 -4419.905} C_VEL
LIN {X 0,Y 531.36,Z 356.751,A -85,B 0,C 180,E1 -4420.864,E2 -4420.864} C_VEL
LIN {X 0,Y 531.626,Z 344.98,A -85,B 0,C 180,E1 -4421.723,E2 -4421.723} C_VEL
LIN {X 0,Y 531.877,Z 333.03,A -85,B 0,C 180,E1 -4422.399,E2 -4422.399} C_VEL
LIN {X 0,Y 532.136,Z 320.662,A -85,B 0,C 180,E1 -4422.926,E2 -4422.926} C_VEL
LIN {X 0,Y 532.082,Z 309.228,A -85,B 0,C 180,E1 -4423.282,E2 -4423.282} C_VEL
LIN {X 0,Y 530.606,Z 300.087,A -85,B 0,C 180,E1 -4423.524,E2 -4423.524} C_VEL
LIN {X 0,Y 530.688,Z 291.402,A -85,B 0,C 180,E1 -4426.542,E2 -4426.542} C_VEL
LIN {X 0,Y 530.774,Z 283.427,A -85,B 0,C 180,E1 -4429.331,E2 -4429.331} C_VEL
LIN {X 0,Y 530.852,Z 275.763,A -85,B 0,C 180,E1 -4432.067,E2 -4432.067} C_VEL
LIN {X 0,Y 531.009,Z 266.614,A -85,B 0,C 180,E1 -4435.45,E2 -4435.45} C_VEL
LIN {X 0,Y 531.127,Z 258.784,A -85,B 0,C 180,E1 -4438.447,E2 -4438.447} C_VEL
LIN {X 0,Y 531.351,Z 251.11,A -85,B 0,C 180,E1 -4441.496,E2 -4441.496} C_VEL
LIN {X 0,Y 531.496,Z 244.638,A -85,B 0,C 180,E1 -4444.192,E2 -4444.192} C_VEL
LIN {X 0,Y 531.453,Z 239.974,A -85,B 0,C 180,E1 -4446.227,E2 -4446.227} C_VEL
LIN {X 0,Y 531.01,Z 237.341,A -85,B 0,C 180,E1 -4447.503,E2 -4447.503} C_VEL
LIN {X 0,Y 530.98,Z 237.348,A -85,B 0,C 180,E1 -4450.432,E2 -4450.432} C_VEL
LIN {X 0,Y 530.965,Z 237.349,A -85,B 0,C 180,E1 -4453.493,E2 -4453.493} C_VEL
LIN {X 0,Y 530.963,Z 237.35,A -85,B 0,C 180,E1 -4456.504,E2 -4456.504} C_VEL
LIN {X 0,Y 531.024,Z 237.343,A -85,B 0,C 180,E1 -4459.57,E2 -4459.57} C_VEL
LIN {X 0,Y 530.974,Z 237.349,A -85,B 0,C 180,E1 -4462.575,E2 -4462.575} C_VEL
LIN {X 0,Y 530.998,Z 237.343,A -85,B 0,C 180,E1 -4465.31,E2 -4465.31} C_VEL
LIN {X 0,Y 530.979,Z 237.346,A -85,B 0,C 180,E1 -4468.032,E2 -4468.032} C_VEL
LIN {X 0,Y 531.003,Z 237.344,A -85,B 0,C 180,E1 -4470.869,E2 -4470.869} C_VEL
LIN {X 0,Y 531.001,Z 237.343,A -85,B 0,C 180,E1 -4473.255,E2 -4473.255} C_VEL
LIN {X 0,Y 530.992,Z 237.346,A -85,B 0,C 180,E1 -4475.957,E2 -4475.957} C_VEL
LIN {X 0,Y 530.994,Z 237.346,A -85,B 0,C 180,E1 -4479.061,E2 -4479.061} C_VEL
LIN {X 0,Y 531.01,Z 237.343,A -85,B 0,C 180,E1 -4482.277,E2 -4482.277} C_VEL
LIN {X 0,Y 531.013,Z 237.343,A -85,B 0,C 180,E1 -4485.435,E2 -4485.435} C_VEL
LIN {X 0,Y 531.04,Z 237.339,A -85,B 0,C 180,E1 -4488.549,E2 -4488.549} C_VEL
LIN {X 0,Y 531.054,Z 237.337,A -85,B 0,C 180,E1 -4491.629,E2 -4491.629} C_VEL
LIN {X 0,Y 531.118,Z 237.329,A -85,B 0,C 180,E1 -4494.684,E2 -4494.684} C_VEL
LIN {X 0,Y 531.131,Z 237.328,A -85,B 0,C 180,E1 -4497.724,E2 -4497.724} C_VEL
LIN {X 0,Y 531.147,Z 237.326,A -85,B 0,C 180,E1 -4500.757,E2 -4500.757} C_VEL
LIN {X 0,Y 531.102,Z 237.332,A -85,B 0,C 180,E1 -4503.033,E2 -4503.033} C_VEL
LIN {X 0,Y 531.077,Z 237.334,A -85,B 0,C 180,E1 -4506.076,E2 -4506.076} C_VEL
LIN {X 0,Y 531.025,Z 237.341,A -85,B 0,C 180,E1 -4509.137,E2 -4509.137} C_VEL
LIN {X 0,Y 530.933,Z 237.394,A -85,B 0,C 180,E1 -4510.679,E2 -4510.679} C_VEL
LIN {X 0,Y 530.913,Z 240.941,A -85,B 0,C 180,E1 -4513.004,E2 -4513.004} C_VEL
LIN {X 0,Y 530.888,Z 244.611,A -85,B 0,C 180,E1 -4515.352,E2 -4515.352} C_VEL
LIN {X 0,Y 530.818,Z 248.381,A -85,B 0,C 180,E1 -4517.728,E2 -4517.728} C_VEL
LIN {X 0,Y 530.718,Z 253.565,A -85,B 0,C 180,E1 -4520.948,E2 -4520.948} C_VEL
LIN {X 0,Y 530.641,Z 258.541,A -85,B 0,C 180,E1 -4523.958,E2 -4523.958} C_VEL
LIN {X 0,Y 530.555,Z 263.228,A -85,B 0,C 180,E1 -4526.767,E2 -4526.767} C_VEL
LIN {X 0,Y 530.468,Z 267.541,A -85,B 0,C 180,E1 -4529.352,E2 -4529.352} C_VEL
LIN {X 0,Y 530.46,Z 272.784,A -85,B 0,C 180,E1 -4532.405,E2 -4532.405} C_VEL
LIN {X 0,Y 530.449,Z 273.063,A -85,B 0,C 180,E1 -4532.56,E2 -4532.56} C_VEL
LIN {X 0,Y 532.26,Z 284.076,A -85,B 0,C 180,E1 -4532.874,E2 -4532.874} C_VEL
LIN {X 0,Y 532.066,Z 296.099,A -85,B 0,C 180,E1 -4533.297,E2 -4533.297} C_VEL
LIN {X 0,Y 531.821,Z 308.296,A -85,B 0,C 180,E1 -4533.882,E2 -4533.882} C_VEL
LIN {X 0,Y 531.602,Z 318.741,A -85,B 0,C 180,E1 -4534.528,E2 -4534.528} C_VEL
LIN {X 0,Y 531.369,Z 329.051,A -85,B 0,C 180,E1 -4535.318,E2 -4535.318} C_VEL
LIN {X 0,Y 531.107,Z 338.196,A -85,B 0,C 180,E1 -4536.179,E2 -4536.179} C_VEL
LIN {X 0,Y 530.93,Z 347.205,A -85,B 0,C 180,E1 -4537.221,E2 -4537.221} C_VEL
LIN {X 0,Y 530.889,Z 348.765,A -85,B 0,C 180,E1 -4537.423,E2 -4537.423} C_VEL
LIN {X 0,Y 530.114,Z 352.441,A -85,B 0,C 180,E1 -4537.917,E2 -4537.917} C_VEL
LIN {X 0,Y 527.152,Z 358.011,A -85,B 0,C 180,E1 -4538.747,E2 -4538.747} C_VEL
LIN {X 0,Y 524.209,Z 362.898,A -85,B 0,C 180,E1 -4539.633,E2 -4539.633} C_VEL
LIN {X 0,Y 523.474,Z 365.503,A -85,B 0,C 180,E1 -4540.209,E2 -4540.209} C_VEL
LIN {X 0,Y 523.425,Z 369.459,A -85,B 0,C 180,E1 -4541.245,E2 -4541.245} C_VEL
LIN {X 0,Y 523.343,Z 372.822,A -85,B 0,C 180,E1 -4542.389,E2 -4542.389} C_VEL
LIN {X 0,Y 523.269,Z 375.169,A -85,B 0,C 180,E1 -4543.51,E2 -4543.51} C_VEL
LIN {X 0,Y 523.295,Z 376.62,A -85,B 0,C 180,E1 -4544.619,E2 -4544.619} C_VEL
LIN {X 0,Y 523.29,Z 377.25,A -85,B 0,C 180,E1 -4545.704,E2 -4545.704} C_VEL
LIN {X 0,Y 523.239,Z 377.131,A -85,B 0,C 180,E1 -4546.764,E2 -4546.764} C_VEL
LIN {X 0,Y 523.302,Z 376.253,A -85,B 0,C 180,E1 -4547.818,E2 -4547.818} C_VEL
LIN {X 0,Y 523.312,Z 373.6,A -85,B 0,C 180,E1 -4549.358,E2 -4549.358} C_VEL
LIN {X 0,Y 523.401,Z 369.362,A -85,B 0,C 180,E1 -4550.87,E2 -4550.87} C_VEL
LIN {X 0,Y 523.513,Z 364.314,A -85,B 0,C 180,E1 -4552.151,E2 -4552.151} C_VEL
LIN {X 0,Y 523.636,Z 357.497,A -85,B 0,C 180,E1 -4553.478,E2 -4553.478} C_VEL
LIN {X 0,Y 523.799,Z 350.752,A -85,B 0,C 180,E1 -4554.529,E2 -4554.529} C_VEL
LIN {X 0,Y 523.995,Z 342.384,A -85,B 0,C 180,E1 -4555.599,E2 -4555.599} C_VEL
LIN {X 0,Y 524.254,Z 333.195,A -85,B 0,C 180,E1 -4556.554,E2 -4556.554} C_VEL
LIN {X 0,Y 524.482,Z 322.058,A -85,B 0,C 180,E1 -4557.487,E2 -4557.487} C_VEL
LIN {X 0,Y 524.717,Z 311.881,A -85,B 0,C 180,E1 -4558.172,E2 -4558.172} C_VEL
LIN {X 0,Y 524.995,Z 300.803,A -85,B 0,C 180,E1 -4558.764,E2 -4558.764} C_VEL
LIN {X 0,Y 525.287,Z 288.236,A -85,B 0,C 180,E1 -4559.263,E2 -4559.263} C_VEL
LIN {X 0,Y 525.139,Z 282.912,A -85,B 0,C 180,E1 -4559.433,E2 -4559.433} C_VEL
LIN {X 0,Y 523.353,Z 273.15,A -85,B 0,C 180,E1 -4559.736,E2 -4559.736} C_VEL
LIN {X 0,Y 523.415,Z 267.83,A -85,B 0,C 180,E1 -4562.838,E2 -4562.838} C_VEL
LIN {X 0,Y 523.428,Z 263.511,A -85,B 0,C 180,E1 -4565.404,E2 -4565.404} C_VEL
LIN {X 0,Y 523.511,Z 259.287,A -85,B 0,C 180,E1 -4567.921,E2 -4567.921} C_VEL
LIN {X 0,Y 523.632,Z 255.222,A -85,B 0,C 180,E1 -4570.395,E2 -4570.395} C_VEL
LIN {X 0,Y 523.668,Z 251.272,A -85,B 0,C 180,E1 -4572.828,E2 -4572.828} C_VEL
LIN {X 0,Y 523.742,Z 247.419,A -85,B 0,C 180,E1 -4575.229,E2 -4575.229} C_VEL
LIN {X 0,Y 523.876,Z 242.432,A -85,B 0,C 180,E1 -4578.391,E2 -4578.391} C_VEL
LIN {X 0,Y 523.838,Z 238.812,A -85,B 0,C 180,E1 -4580.736,E2 -4580.736} C_VEL
LIN {X 0,Y 523.913,Z 238.223,A -85,B 0,C 180,E1 -4581.515,E2 -4581.515} C_VEL
LIN {X 0,Y 524.036,Z 238.211,A -85,B 0,C 180,E1 -4583.841,E2 -4583.841} C_VEL
LIN {X 0,Y 524.064,Z 238.208,A -85,B 0,C 180,E1 -4586.925,E2 -4586.925} C_VEL
LIN {X 0,Y 524.102,Z 238.202,A -85,B 0,C 180,E1 -4590,E2 -4590} C_VEL
LIN {X 0,Y 524.065,Z 238.209,A -85,B 0,C 180,E1 -4593.075,E2 -4593.075} C_VEL
LIN {X 0,Y 524.036,Z 238.21,A -85,B 0,C 180,E1 -4596.159,E2 -4596.159} C_VEL
LIN {X 0,Y 523.995,Z 238.216,A -85,B 0,C 180,E1 -4599.262,E2 -4599.262} C_VEL
LIN {X 0,Y 524.014,Z 238.215,A -85,B 0,C 180,E1 -4601.751,E2 -4601.751} C_VEL
LIN {X 0,Y 523.981,Z 238.218,A -85,B 0,C 180,E1 -4605.053,E2 -4605.053} C_VEL
LIN {X 0,Y 523.954,Z 238.221,A -85,B 0,C 180,E1 -4607.969,E2 -4607.969} C_VEL
LIN {X 0,Y 523.963,Z 238.219,A -85,B 0,C 180,E1 -4610.41,E2 -4610.41} C_VEL
LIN {X 0,Y 523.934,Z 238.222,A -85,B 0,C 180,E1 -4612.892,E2 -4612.892} C_VEL
LIN {X 0,Y 523.975,Z 238.22,A -85,B 0,C 180,E1 -4616.021,E2 -4616.021} C_VEL
LIN {X 0,Y 523.94,Z 238.221,A -85,B 0,C 180,E1 -4618.874,E2 -4618.874} C_VEL
LIN {X 0,Y 523.922,Z 238.224,A -85,B 0,C 180,E1 -4621.544,E2 -4621.544} C_VEL
LIN {X 0,Y 523.932,Z 238.225,A -85,B 0,C 180,E1 -4624.29,E2 -4624.29} C_VEL
LIN {X 0,Y 523.9,Z 238.228,A -85,B 0,C 180,E1 -4627.132,E2 -4627.132} C_VEL
LIN {X 0,Y 523.957,Z 238.221,A -85,B 0,C 180,E1 -4630.134,E2 -4630.134} C_VEL
LIN {X 0,Y 523.915,Z 238.226,A -85,B 0,C 180,E1 -4633.167,E2 -4633.167} C_VEL
LIN {X 0,Y 523.93,Z 238.223,A -85,B 0,C 180,E1 -4635.773,E2 -4635.773} C_VEL
LIN {X 0,Y 523.951,Z 238.223,A -85,B 0,C 180,E1 -4638.91,E2 -4638.91} C_VEL
LIN {X 0,Y 523.906,Z 238.226,A -85,B 0,C 180,E1 -4641.899,E2 -4641.899} C_VEL
LIN {X 0,Y 523.927,Z 238.226,A -85,B 0,C 180,E1 -4644.909,E2 -4644.909} C_VEL
LIN {X 0,Y 523.932,Z 238.222,A -85,B 0,C 180,E1 -4647.679,E2 -4647.679} C_VEL
LIN {X 0,Y 523.959,Z 238.221,A -85,B 0,C 180,E1 -4650.674,E2 -4650.674} C_VEL
LIN {X 0,Y 523.968,Z 238.217,A -85,B 0,C 180,E1 -4653.729,E2 -4653.729} C_VEL
LIN {X 0,Y 523.926,Z 238.223,A -85,B 0,C 180,E1 -4656.272,E2 -4656.272} C_VEL
LIN {X 0,Y 523.938,Z 238.223,A -85,B 0,C 180,E1 -4658.768,E2 -4658.768} C_VEL
LIN {X 0,Y 523.945,Z 238.222,A -85,B 0,C 180,E1 -4661.222,E2 -4661.222} C_VEL
LIN {X 0,Y 523.931,Z 238.223,A -85,B 0,C 180,E1 -4663.64,E2 -4663.64} C_VEL
LIN {X 0,Y 523.93,Z 238.223,A -85,B 0,C 180,E1 -4666.029,E2 -4666.029} C_VEL
LIN {X 0,Y 524.003,Z 238.214,A -85,B 0,C 180,E1 -4668.395,E2 -4668.395} C_VEL
LIN {X 0,Y 524,Z 238.215,A -85,B 0,C 180,E1 -4671.517,E2 -4671.517} C_VEL
LIN {X 0,Y 524.076,Z 238.207,A -85,B 0,C 180,E1 -4674.615,E2 -4674.615} C_VEL
LIN {X 0,Y 524.105,Z 238.201,A -85,B 0,C 180,E1 -4677.695,E2 -4677.695} C_VEL
LIN {X 0,Y 524.119,Z 238.202,A -85,B 0,C 180,E1 -4680.769,E2 -4680.769} C_VEL
LIN {X 0,Y 524.067,Z 238.207,A -85,B 0,C 180,E1 -4683.076,E2 -4683.076} C_VEL
LIN {X 0,Y 524.039,Z 238.21,A -85,B 0,C 180,E1 -4686.16,E2 -4686.16} C_VEL
LIN {X 0,Y 523.992,Z 238.217,A -85,B 0,C 180,E1 -4689.263,E2 -4689.263} C_VEL
LIN {X 0,Y 524.019,Z 238.214,A -85,B 0,C 180,E1 -4691.752,E2 -4691.752} C_VEL
LIN {X 0,Y 523.988,Z 238.217,A -85,B 0,C 180,E1 -4695.053,E2 -4695.053} C_VEL
LIN {X 0,Y 523.959,Z 238.22,A -85,B 0,C 180,E1 -4697.97,E2 -4697.97} C_VEL
LIN {X 0,Y 523.968,Z 238.218,A -85,B 0,C 180,E1 -4700.411,E2 -4700.411} C_VEL
LIN {X 0,Y 523.913,Z 238.225,A -85,B 0,C 180,E1 -4702.894,E2 -4702.894} C_VEL
LIN {X 0,Y 523.949,Z 238.221,A -85,B 0,C 180,E1 -4705.42,E2 -4705.42} C_VEL
LIN {X 0,Y 523.967,Z 238.219,A -85,B 0,C 180,E1 -4708,E2 -4708} C_VEL
LIN {X 0,Y 523.941,Z 238.223,A -85,B 0,C 180,E1 -4710.856,E2 -4710.856} C_VEL
LIN {X 0,Y 523.929,Z 238.223,A -85,B 0,C 180,E1 -4713.731,E2 -4713.731} C_VEL
LIN {X 0,Y 523.918,Z 238.224,A -85,B 0,C 180,E1 -4716.405,E2 -4716.405} C_VEL
LIN {X 0,Y 523.921,Z 238.226,A -85,B 0,C 180,E1 -4719.085,E2 -4719.085} C_VEL
LIN {X 0,Y 523.952,Z 238.219,A -85,B 0,C 180,E1 -4722.12,E2 -4722.12} C_VEL
LIN {X 0,Y 523.949,Z 238.223,A -85,B 0,C 180,E1 -4725.31,E2 -4725.31} C_VEL
LIN {X 0,Y 523.961,Z 238.221,A -85,B 0,C 180,E1 -4728.69,E2 -4728.69} C_VEL
LIN {X 0,Y 523.924,Z 238.224,A -85,B 0,C 180,E1 -4731.9,E2 -4731.9} C_VEL
LIN {X 0,Y 523.952,Z 238.25,A -85,B 0,C 180,E1 -4732.46,E2 -4732.46} C_VEL
LIN {X 0,Y 524.56,Z 242.469,A -85,B 0,C 180,E1 -4734.353,E2 -4734.353} C_VEL
LIN {X 0,Y 524.463,Z 249.051,A -85,B 0,C 180,E1 -4737.132,E2 -4737.132} C_VEL
LIN {X 0,Y 524.257,Z 256.75,A -85,B 0,C 180,E1 -4740.264,E2 -4740.264} C_VEL
LIN {X 0,Y 524.019,Z 264.49,A -85,B 0,C 180,E1 -4743.302,E2 -4743.302} C_VEL
LIN {X 0,Y 523.891,Z 272.258,A -85,B 0,C 180,E1 -4746.269,E2 -4746.269} C_VEL
LIN {X 0,Y 523.789,Z 280.194,A -85,B 0,C 180,E1 -4749.172,E2 -4749.172} C_VEL
LIN {X 0,Y 523.706,Z 288.083,A -85,B 0,C 180,E1 -4752.022,E2 -4752.022} C_VEL
LIN {X 0,Y 523.589,Z 297.007,A -85,B 0,C 180,E1 -4755.225,E2 -4755.225} C_VEL
LIN {X 0,Y 523.55,Z 299.996,A -85,B 0,C 180,E1 -4756.29,E2 -4756.29} C_VEL
LIN {X 0,Y 525.367,Z 312.379,A -85,B 0,C 180,E1 -4756.634,E2 -4756.634} C_VEL
LIN {X 0,Y 525.115,Z 325.454,A -85,B 0,C 180,E1 -4757.095,E2 -4757.095} C_VEL
LIN {X 0,Y 524.83,Z 337.744,A -85,B 0,C 180,E1 -4757.694,E2 -4757.694} C_VEL
LIN {X 0,Y 524.526,Z 349.02,A -85,B 0,C 180,E1 -4758.406,E2 -4758.406} C_VEL
LIN {X 0,Y 524.308,Z 359.956,A -85,B 0,C 180,E1 -4759.282,E2 -4759.282} C_VEL
LIN {X 0,Y 524.037,Z 368.867,A -85,B 0,C 180,E1 -4760.154,E2 -4760.154} C_VEL
LIN {X 0,Y 523.821,Z 378.549,A -85,B 0,C 180,E1 -4761.319,E2 -4761.319} C_VEL
LIN {X 0,Y 523.63,Z 386.258,A -85,B 0,C 180,E1 -4762.481,E2 -4762.481} C_VEL
LIN {X 0,Y 523.494,Z 393.36,A -85,B 0,C 180,E1 -4763.834,E2 -4763.834} C_VEL
LIN {X 0,Y 523.384,Z 398.083,A -85,B 0,C 180,E1 -4764.993,E2 -4764.993} C_VEL
LIN {X 0,Y 523.444,Z 401.696,A -85,B 0,C 180,E1 -4766.151,E2 -4766.151} C_VEL
LIN {X 0,Y 523.368,Z 403.555,A -85,B 0,C 180,E1 -4766.921,E2 -4766.921} C_VEL
LIN {X 0,Y 523.335,Z 404.95,A -85,B 0,C 180,E1 -4767.691,E2 -4767.691} C_VEL
LIN {X 0,Y 523.25,Z 406.552,A -85,B 0,C 180,E1 -4769.23,E2 -4769.23} C_VEL
LIN {X 0,Y 523.246,Z 406.767,A -85,B 0,C 180,E1 -4770,E2 -4770} C_VEL
LIN {X 0,Y 523.275,Z 405.943,A -85,B 0,C 180,E1 -4771.539,E2 -4771.539} C_VEL
LIN {X 0,Y 523.335,Z 404.949,A -85,B 0,C 180,E1 -4772.309,E2 -4772.309} C_VEL
LIN {X 0,Y 523.368,Z 403.552,A -85,B 0,C 180,E1 -4773.079,E2 -4773.079} C_VEL
LIN {X 0,Y 523.425,Z 400.615,A -85,B 0,C 180,E1 -4774.235,E2 -4774.235} C_VEL
LIN {X 0,Y 523.461,Z 396.637,A -85,B 0,C 180,E1 -4775.393,E2 -4775.393} C_VEL
LIN {X 0,Y 523.518,Z 391.405,A -85,B 0,C 180,E1 -4776.575,E2 -4776.575} C_VEL
LIN {X 0,Y 523.652,Z 385.067,A -85,B 0,C 180,E1 -4777.713,E2 -4777.713} C_VEL
LIN {X 0,Y 523.836,Z 377.023,A -85,B 0,C 180,E1 -4778.875,E2 -4778.875} C_VEL
LIN {X 0,Y 524.036,Z 368.823,A -85,B 0,C 180,E1 -4779.845,E2 -4779.845} C_VEL
LIN {X 0,Y 524.328,Z 358.825,A -85,B 0,C 180,E1 -4780.816,E2 -4780.816} C_VEL
LIN {X 0,Y 524.608,Z 347.631,A -85,B 0,C 180,E1 -4781.683,E2 -4781.683} C_VEL
LIN {X 0,Y 524.829,Z 336.467,A -85,B 0,C 180,E1 -4782.372,E2 -4782.372} C_VEL
LIN {X 0,Y 525.132,Z 324.223,A -85,B 0,C 180,E1 -4782.954,E2 -4782.954} C_VEL
LIN {X 0,Y 525.282,Z 310.889,A -85,B 0,C 180,E1 -4783.405,E2 -4783.405} C_VEL
LIN {X 0,Y 523.549,Z 299.865,A -85,B 0,C 180,E1 -4783.71,E2 -4783.71} C_VEL
LIN {X 0,Y 523.634,Z 291.212,A -85,B 0,C 180,E1 -4786.772,E2 -4786.772} C_VEL
LIN {X 0,Y 523.719,Z 281.986,A -85,B 0,C 180,E1 -4790.055,E2 -4790.055} C_VEL
LIN {X 0,Y 523.842,Z 274.239,A -85,B 0,C 180,E1 -4792.896,E2 -4792.896} C_VEL
LIN {X 0,Y 523.971,Z 265.987,A -85,B 0,C 180,E1 -4796.016,E2 -4796.016} C_VEL
LIN {X 0,Y 524.196,Z 257.412,A -85,B 0,C 180,E1 -4799.369,E2 -4799.369} C_VEL
LIN {X 0,Y 524.367,Z 249.972,A -85,B 0,C 180,E1 -4802.419,E2 -4802.419} C_VEL
LIN {X 0,Y 524.567,Z 243.544,A -85,B 0,C 180,E1 -4805.188,E2 -4805.188} C_VEL
LIN {X 0,Y 524.397,Z 240.705,A -85,B 0,C 180,E1 -4806.474,E2 -4806.474} C_VEL
LIN {X 0,Y 523.947,Z 238.221,A -85,B 0,C 180,E1 -4807.683,E2 -4807.683} C_VEL
LIN {X 0,Y 523.941,Z 238.224,A -85,B 0,C 180,E1 -4811.091,E2 -4811.091} C_VEL
LIN {X 0,Y 523.94,Z 238.223,A -85,B 0,C 180,E1 -4814.227,E2 -4814.227} C_VEL
LIN {X 0,Y 523.92,Z 238.226,A -85,B 0,C 180,E1 -4816.832,E2 -4816.832} C_VEL
LIN {X 0,Y 523.976,Z 238.219,A -85,B 0,C 180,E1 -4819.922,E2 -4819.922} C_VEL
LIN {X 0,Y 523.915,Z 238.226,A -85,B 0,C 180,E1 -4822.868,E2 -4822.868} C_VEL
LIN {X 0,Y 523.941,Z 238.225,A -85,B 0,C 180,E1 -4825.71,E2 -4825.71} C_VEL
LIN {X 0,Y 523.929,Z 238.224,A -85,B 0,C 180,E1 -4828.456,E2 -4828.456} C_VEL
LIN {X 0,Y 523.947,Z 238.222,A -85,B 0,C 180,E1 -4831.125,E2 -4831.125} C_VEL
LIN {X 0,Y 523.979,Z 238.22,A -85,B 0,C 180,E1 -4833.979,E2 -4833.979} C_VEL
LIN {X 0,Y 523.931,Z 238.224,A -85,B 0,C 180,E1 -4836.27,E2 -4836.27} C_VEL
LIN {X 0,Y 523.94,Z 238.223,A -85,B 0,C 180,E1 -4838.766,E2 -4838.766} C_VEL
LIN {X 0,Y 523.948,Z 238.223,A -85,B 0,C 180,E1 -4841.22,E2 -4841.22} C_VEL
LIN {X 0,Y 523.934,Z 238.223,A -85,B 0,C 180,E1 -4843.638,E2 -4843.638} C_VEL
LIN {X 0,Y 523.935,Z 238.224,A -85,B 0,C 180,E1 -4846.027,E2 -4846.027} C_VEL
LIN {X 0,Y 524.005,Z 238.216,A -85,B 0,C 180,E1 -4848.393,E2 -4848.393} C_VEL
LIN {X 0,Y 524.002,Z 238.216,A -85,B 0,C 180,E1 -4851.515,E2 -4851.515} C_VEL
LIN {X 0,Y 524.078,Z 238.206,A -85,B 0,C 180,E1 -4854.613,E2 -4854.613} C_VEL
LIN {X 0,Y 524.103,Z 238.203,A -85,B 0,C 180,E1 -4857.694,E2 -4857.694} C_VEL
LIN {X 0,Y 524.117,Z 238.202,A -85,B 0,C 180,E1 -4860.767,E2 -4860.767} C_VEL
LIN {X 0,Y 524.068,Z 238.208,A -85,B 0,C 180,E1 -4863.074,E2 -4863.074} C_VEL
LIN {X 0,Y 524.039,Z 238.211,A -85,B 0,C 180,E1 -4866.158,E2 -4866.158} C_VEL
LIN {X 0,Y 523.989,Z 238.217,A -85,B 0,C 180,E1 -4869.261,E2 -4869.261} C_VEL
LIN {X 0,Y 523.908,Z 238.536,A -85,B 0,C 180,E1 -4870.824,E2 -4870.824} C_VEL
LIN {X 0,Y 523.879,Z 242.105,A -85,B 0,C 180,E1 -4873.182,E2 -4873.182} C_VEL
LIN {X 0,Y 523.828,Z 245.782,A -85,B 0,C 180,E1 -4875.564,E2 -4875.564} C_VEL
LIN {X 0,Y 523.751,Z 249.575,A -85,B 0,C 180,E1 -4877.975,E2 -4877.975} C_VEL
LIN {X 0,Y 523.662,Z 253.477,A -85,B 0,C 180,E1 -4880.421,E2 -4880.421} C_VEL
LIN {X 0,Y 523.582,Z 257.471,A -85,B 0,C 180,E1 -4882.908,E2 -4882.908} C_VEL
LIN {X 0,Y 523.534,Z 262.459,A -85,B 0,C 180,E1 -4885.921,E2 -4885.921} C_VEL
LIN {X 0,Y 523.473,Z 265.919,A -85,B 0,C 180,E1 -4888.027,E2 -4888.027} C_VEL
LIN {X 0,Y 523.394,Z 270.51,A -85,B 0,C 180,E1 -4890.756,E2 -4890.756} C_VEL
LIN {X 0,Y 523.386,Z 273.262,A -85,B 0,C 180,E1 -4892.366,E2 -4892.366} C_VEL
LIN {X 0,Y 525.342,Z 284.5,A -85,B 0,C 180,E1 -4892.706,E2 -4892.706} C_VEL
LIN {X 0,Y 525.138,Z 297.103,A -85,B 0,C 180,E1 -4893.162,E2 -4893.162} C_VEL
LIN {X 0,Y 524.859,Z 309.948,A -85,B 0,C 180,E1 -4893.802,E2 -4893.802} C_VEL
LIN {X 0,Y 524.613,Z 320.323,A -85,B 0,C 180,E1 -4894.471,E2 -4894.471} C_VEL
LIN {X 0,Y 524.336,Z 330.759,A -85,B 0,C 180,E1 -4895.311,E2 -4895.311} C_VEL
LIN {X 0,Y 524.064,Z 340.611,A -85,B 0,C 180,E1 -4896.29,E2 -4896.29} C_VEL
LIN {X 0,Y 523.851,Z 349.615,A -85,B 0,C 180,E1 -4897.394,E2 -4897.394} C_VEL
LIN {X 0,Y 523.66,Z 356.863,A -85,B 0,C 180,E1 -4898.497,E2 -4898.497} C_VEL
LIN {X 0,Y 523.525,Z 363.814,A -85,B 0,C 180,E1 -4899.827,E2 -4899.827} C_VEL
LIN {X 0,Y 523.474,Z 365.503,A -85,B 0,C 180,E1 -4900.209,E2 -4900.209} C_VEL
LIN {X 0,Y 522.731,Z 367.909,A -85,B 0,C 180,E1 -4900.798,E2 -4900.798} C_VEL
LIN {X 0,Y 519.773,Z 371.32,A -85,B 0,C 180,E1 -4901.771,E2 -4901.771} C_VEL
LIN {X 0,Y 517.313,Z 373.508,A -85,B 0,C 180,E1 -4902.573,E2 -4902.573} C_VEL
LIN {X 0,Y 516.26,Z 374.864,A -85,B 0,C 180,E1 -4903.203,E2 -4903.203} C_VEL
LIN {X 0,Y 516.175,Z 375.193,A -85,B 0,C 180,E1 -4903.418,E2 -4903.418} C_VEL
LIN {X 0,Y 516.188,Z 376.11,A -85,B 0,C 180,E1 -4903.976,E2 -4903.976} C_VEL
LIN {X 0,Y 516.195,Z 377.182,A -85,B 0,C 180,E1 -4905.069,E2 -4905.069} C_VEL
LIN {X 0,Y 516.171,Z 377.491,A -85,B 0,C 180,E1 -4906.187,E2 -4906.187} C_VEL
LIN {X 0,Y 516.168,Z 376.977,A -85,B 0,C 180,E1 -4907.326,E2 -4907.326} C_VEL
LIN {X 0,Y 516.201,Z 375.563,A -85,B 0,C 180,E1 -4908.486,E2 -4908.486} C_VEL
LIN {X 0,Y 516.238,Z 373.181,A -85,B 0,C 180,E1 -4909.672,E2 -4909.672} C_VEL
LIN {X 0,Y 516.33,Z 369.729,A -85,B 0,C 180,E1 -4910.88,E2 -4910.88} C_VEL
LIN {X 0,Y 516.446,Z 364.477,A -85,B 0,C 180,E1 -4912.239,E2 -4912.239} C_VEL
LIN {X 0,Y 516.596,Z 357.6,A -85,B 0,C 180,E1 -4913.593,E2 -4913.593} C_VEL
LIN {X 0,Y 516.76,Z 350.657,A -85,B 0,C 180,E1 -4914.685,E2 -4914.685} C_VEL
LIN {X 0,Y 517.01,Z 341.571,A -85,B 0,C 180,E1 -4915.841,E2 -4915.841} C_VEL
LIN {X 0,Y 517.315,Z 331.677,A -85,B 0,C 180,E1 -4916.852,E2 -4916.852} C_VEL
LIN {X 0,Y 517.522,Z 321.516,A -85,B 0,C 180,E1 -4917.697,E2 -4917.697} C_VEL
LIN {X 0,Y 517.804,Z 310.681,A -85,B 0,C 180,E1 -4918.421,E2 -4918.421} C_VEL
LIN {X 0,Y 518.119,Z 298.874,A -85,B 0,C 180,E1 -4919.03,E2 -4919.03} C_VEL
LIN {X 0,Y 518.468,Z 285.538,A -85,B 0,C 180,E1 -4919.533,E2 -4919.533} C_VEL
LIN {X 0,Y 516.277,Z 273.341,A -85,B 0,C 180,E1 -4919.927,E2 -4919.927} C_VEL
LIN {X 0,Y 516.303,Z 269.073,A -85,B 0,C 180,E1 -4922.432,E2 -4922.432} C_VEL
LIN {X 0,Y 516.352,Z 264.696,A -85,B 0,C 180,E1 -4925.044,E2 -4925.044} C_VEL
LIN {X 0,Y 516.463,Z 260.276,A -85,B 0,C 180,E1 -4927.716,E2 -4927.716} C_VEL
LIN {X 0,Y 516.555,Z 256.359,A -85,B 0,C 180,E1 -4930.115,E2 -4930.115} C_VEL
LIN {X 0,Y 516.592,Z 252.381,A -85,B 0,C 180,E1 -4932.585,E2 -4932.585} C_VEL
LIN {X 0,Y 516.686,Z 247.249,A -85,B 0,C 180,E1 -4935.828,E2 -4935.828} C_VEL
LIN {X 0,Y 516.83,Z 242.271,A -85,B 0,C 180,E1 -4939.026,E2 -4939.026} C_VEL
